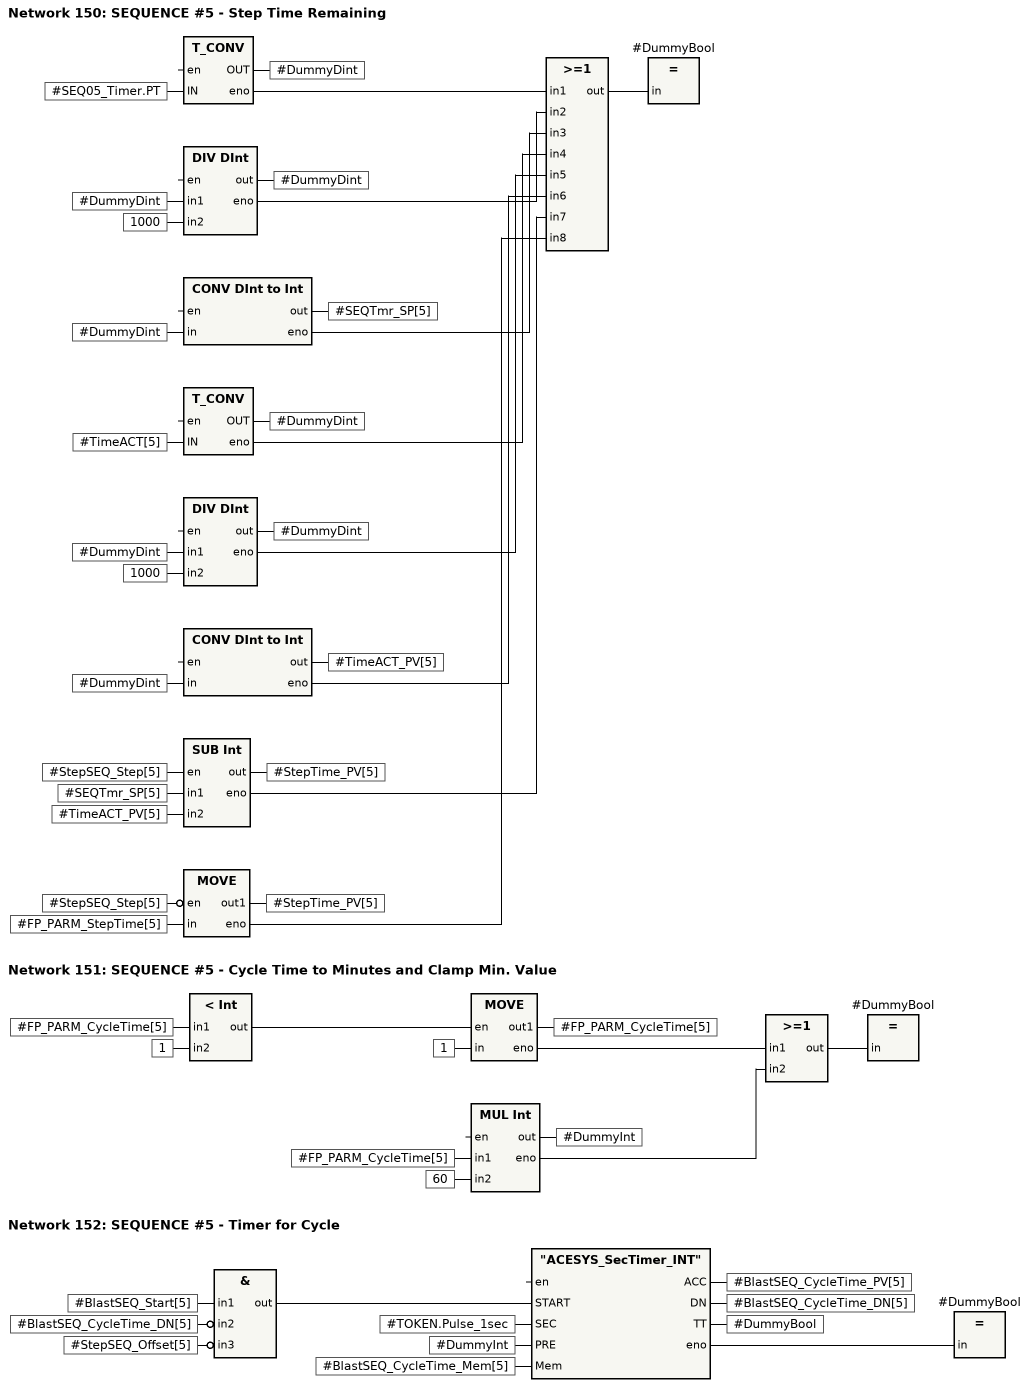
   // ENO of a box is taken as its EN; it also drops when the box reports an error
   #DummyDint := T_CONV(IN := #SEQ05_Timer.PT);
   #DummyDint := #DummyDint / 1000;
   #SEQTmr_SP[5] := DINT_TO_INT(#DummyDint);
   #DummyDint := T_CONV(IN := #TimeACT[5]);
   #DummyDint := #DummyDint / 1000;
   #TimeACT_PV[5] := DINT_TO_INT(#DummyDint);
   IF #StepSEQ_Step[5] THEN #StepTime_PV[5] := #SEQTmr_SP[5] - #TimeACT_PV[5]; END_IF;
   IF NOT #StepSEQ_Step[5] THEN #StepTime_PV[5] := #FP_PARM_StepTime[5]; END_IF;
   #DummyBool := TRUE OR TRUE OR TRUE OR TRUE OR TRUE OR TRUE OR #StepSEQ_Step[5] OR NOT #StepSEQ_Step[5];
END_REGION

REGION Network 151: SEQUENCE #5 - Cycle Time to Minutes and Clamp Min. Value
   // ENO of a box is taken as its EN; it also drops when the box reports an error
   #_w1 := #FP_PARM_CycleTime[5] < 1;
   IF #_w1 THEN #FP_PARM_CycleTime[5] := 1; END_IF;
   #DummyInt := #FP_PARM_CycleTime[5] * 60;
   #DummyBool := #_w1 OR TRUE;
END_REGION

REGION Network 152: SEQUENCE #5 - Timer for Cycle
   "ACESYS_SecTimer_INT"(START := #BlastSEQ_Start[5] AND NOT #BlastSEQ_CycleTime_DN[5] AND NOT #StepSEQ_Offset[5],
                         SEC := #TOKEN.Pulse_1sec,
                         PRE := #DummyInt,
                         Mem := #BlastSEQ_CycleTime_Mem[5],
                         ACC => #BlastSEQ_CycleTime_PV[5],
                         DN => #BlastSEQ_CycleTime_DN[5],
                         TT => #DummyBool,
                         ENO => #_w1);
   #DummyBool := #_w1;
END_REGION

REGION Network 153: SEQUENCE #6 - Enable and Start
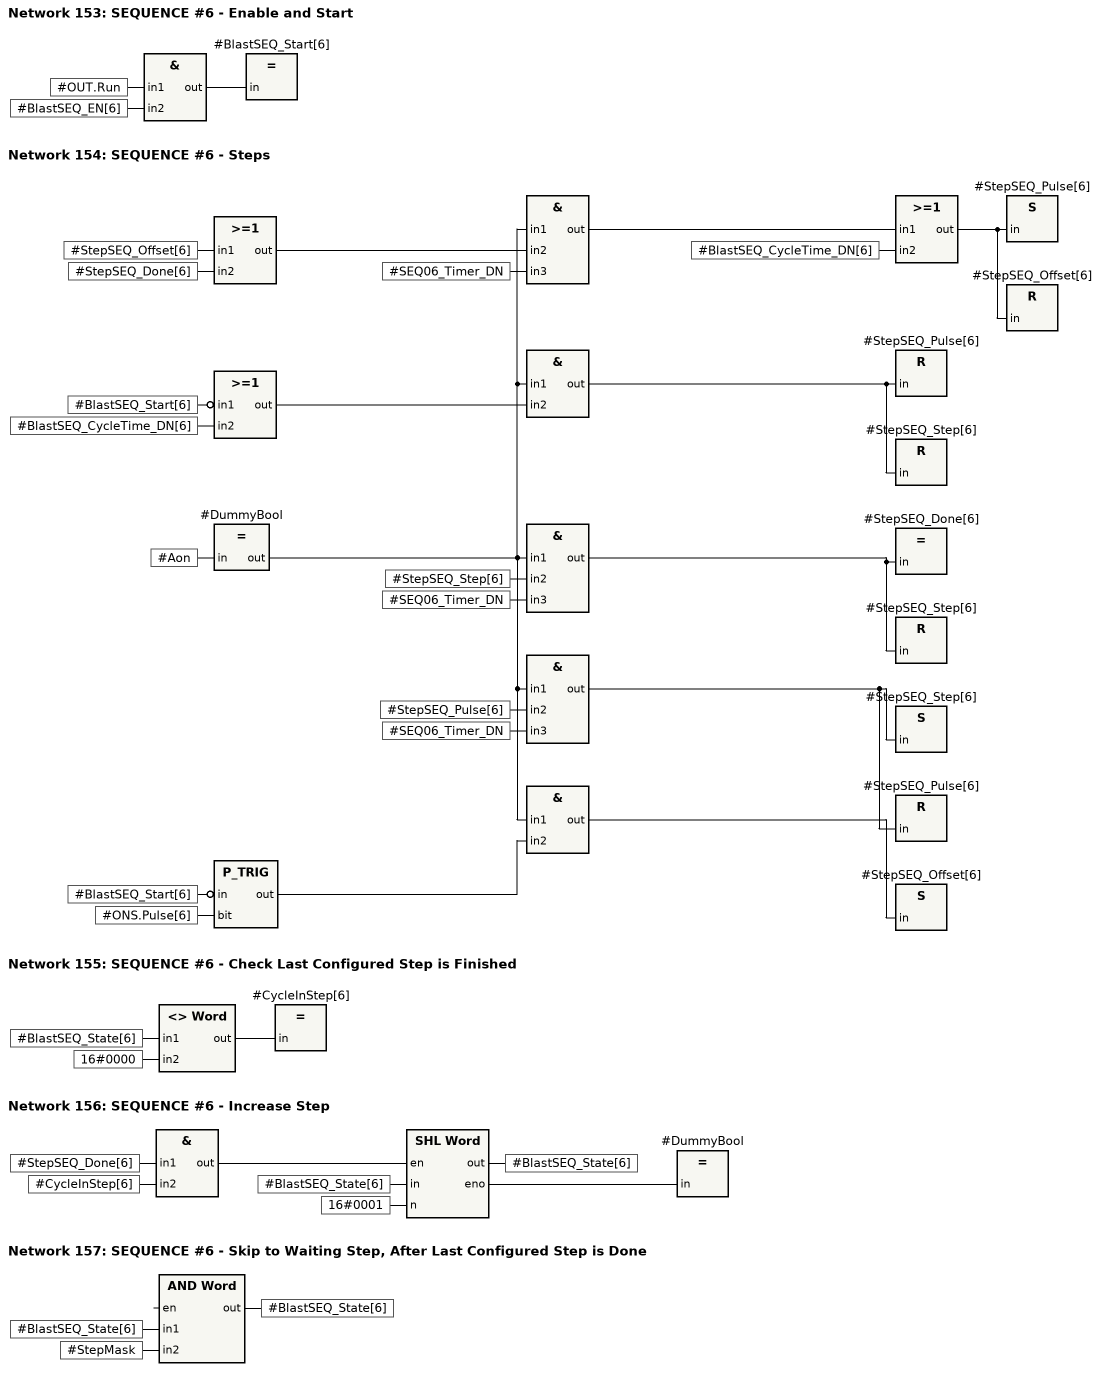
   #BlastSEQ_Start[6] := #OUT.Run AND #BlastSEQ_EN[6];
END_REGION

REGION Network 154: SEQUENCE #6 - Steps
   // Build 002 - 25.Apr.2020 (MIA-US): Replace timer's Q output with tag
   // 
   // ***
   // SEQUENCE 06 LOGIC
   // ***
   // 
   // ***Blaster Sequence***
   // 16#0001 = BQ01
   // 16#0002 = BQ02
   //   -||-
   // 16#4000 = BQ15
   // 16#8000 = BQ16
   // 16#0000 = Cycle Time
   // 
   // ***Step Sequence***
   // - Offset Time
   // - Pulse Time
   // - Step Time
   // - Step Completed
   #DummyBool := #Aon;
   IF #Aon AND (NOT #BlastSEQ_Start[6] OR #BlastSEQ_CycleTime_DN[6]) THEN
       #StepSEQ_Pulse[6] := FALSE;
       #StepSEQ_Step[6] := FALSE;
   END_IF;
   #StepSEQ_Done[6] := #Aon AND #StepSEQ_Step[6] AND #SEQ06_Timer_DN;
   IF #Aon AND #StepSEQ_Step[6] AND #SEQ06_Timer_DN THEN #StepSEQ_Step[6] := FALSE; END_IF;
   IF #Aon AND #StepSEQ_Pulse[6] AND #SEQ06_Timer_DN THEN
       #StepSEQ_Step[6] := TRUE;
       #StepSEQ_Pulse[6] := FALSE;
   END_IF;
   IF (#Aon AND (#StepSEQ_Offset[6] OR #StepSEQ_Done[6]) AND #SEQ06_Timer_DN) OR #BlastSEQ_CycleTime_DN[6] THEN
       #StepSEQ_Pulse[6] := TRUE;
       #StepSEQ_Offset[6] := FALSE;
   END_IF;
   #_w1 := NOT #BlastSEQ_Start[6] AND NOT #ONS.Pulse[6];   // rising edge
   #ONS.Pulse[6] := NOT #BlastSEQ_Start[6];
   IF #Aon AND #_w1 THEN #StepSEQ_Offset[6] := TRUE; END_IF;
END_REGION

REGION Network 155: SEQUENCE #6 - Check Last Configured Step is Finished
   // 16#0000 is the waiting state
   #CycleInStep[6] := #BlastSEQ_State[6] <> 16#0000;
END_REGION

REGION Network 156: SEQUENCE #6 - Increase Step
   // Set next step by shifting one bit to the left in the sequence status
   // ENO of a box is taken as its EN; it also drops when the box reports an error
   #_w1 := #StepSEQ_Done[6] AND #CycleInStep[6];
   IF #_w1 THEN #BlastSEQ_State[6] := SHL(IN := #BlastSEQ_State[6], N := 16#0001); END_IF;
   #DummyBool := #_w1;
END_REGION

REGION Network 157: SEQUENCE #6 - Skip to Waiting Step, After Last Configured Step is Done
   // Sequence Status will become 16#0000 once the shifting bit moves into the unconfigured steps (0 in Step Mask)
   #BlastSEQ_State[6] := #BlastSEQ_State[6] AND #StepMask;
END_REGION

REGION Network 158: SEQUENCE #6 - Offset Step
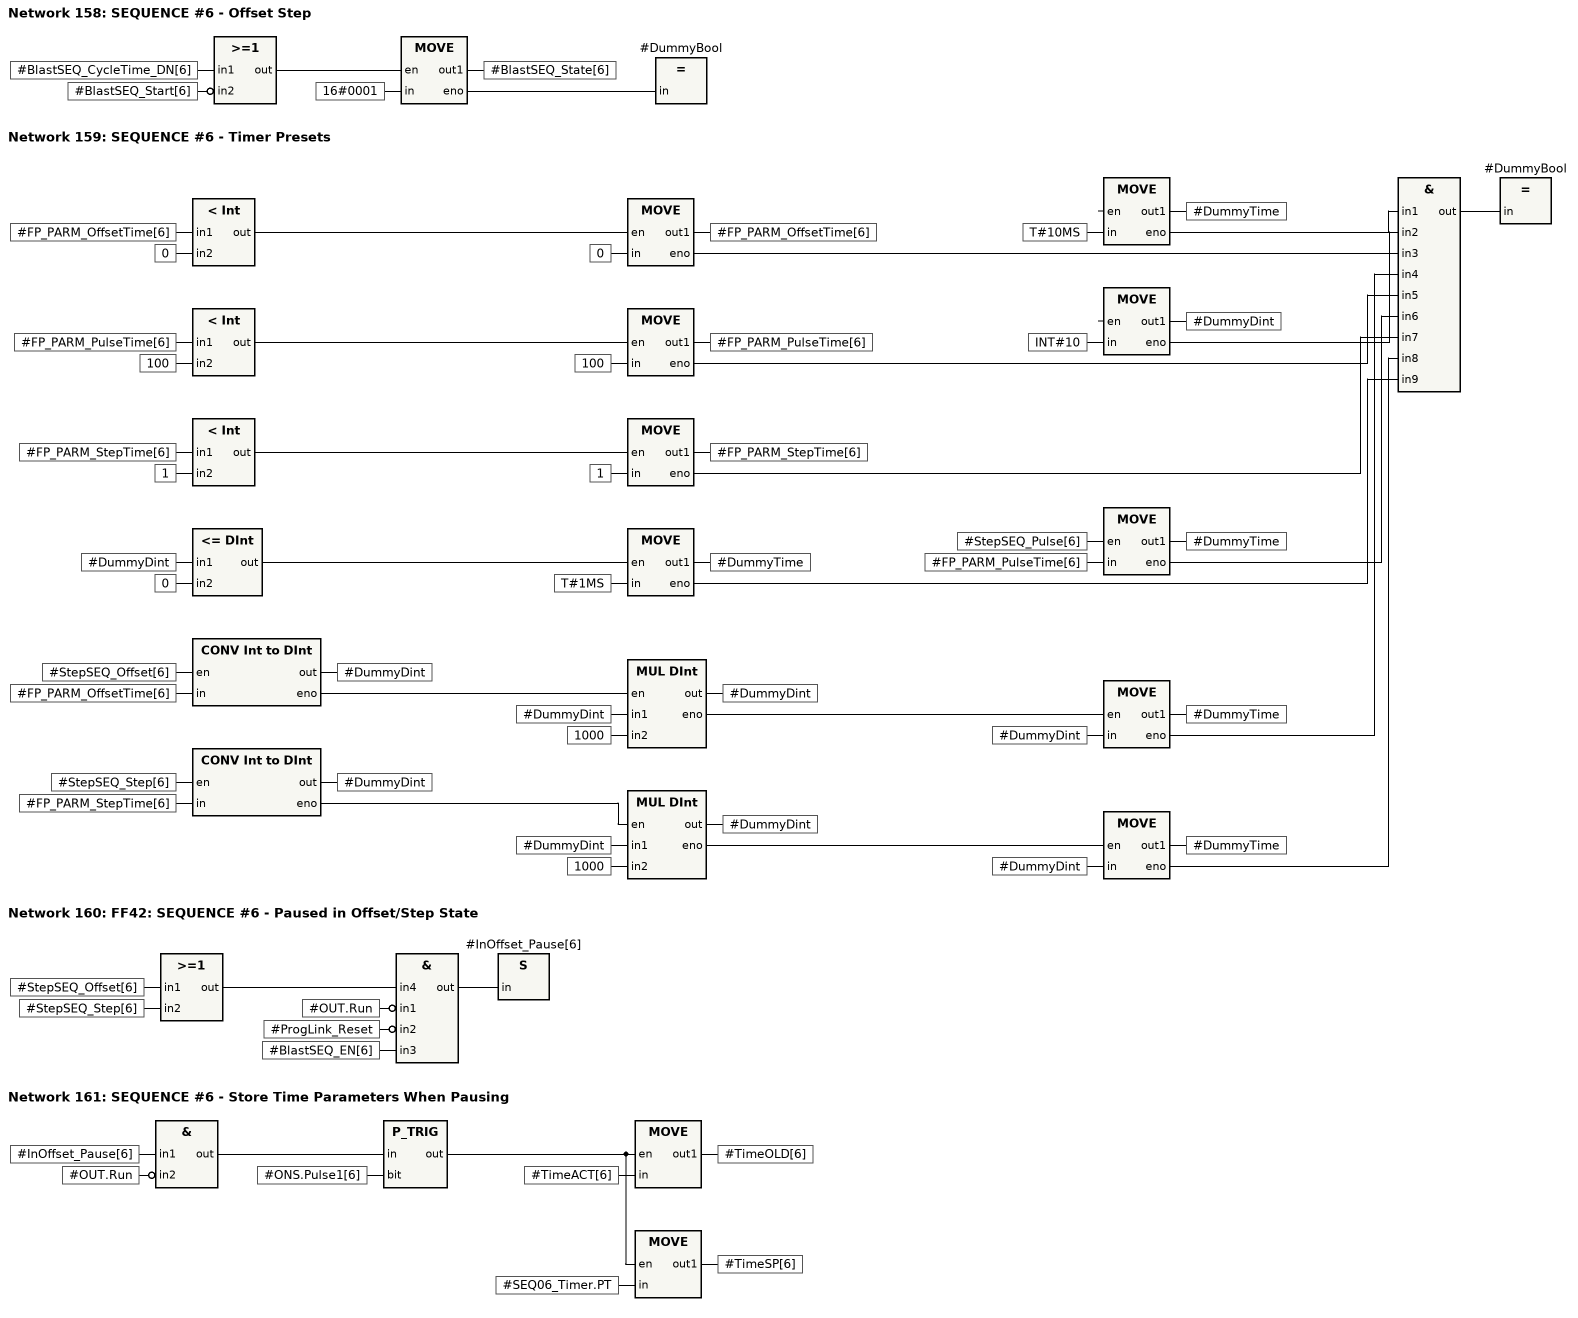
   // ENO of a box is taken as its EN; it also drops when the box reports an error
   #_w1 := #BlastSEQ_CycleTime_DN[6] OR NOT #BlastSEQ_Start[6];
   IF #_w1 THEN #BlastSEQ_State[6] := 16#0001; END_IF;
   #DummyBool := #_w1;
END_REGION

REGION Network 159: SEQUENCE #6 - Timer Presets
   // *Convert Offset Time to minutes and clamp minimum value
   // 
   // *Convert Pulse Time to ms and clamp minimum value
   // 
   // *Convert Step Time to seconds and clamp minimum value
   // ENO of a box is taken as its EN; it also drops when the box reports an error
   #DummyTime := T#10MS;
   #DummyDint := INT#10;
   #_w1 := #FP_PARM_OffsetTime[6] < 0;
   IF #_w1 THEN #FP_PARM_OffsetTime[6] := 0; END_IF;
   IF #StepSEQ_Offset[6] THEN
       #DummyDint := INT_TO_DINT(#FP_PARM_OffsetTime[6]);
       #DummyDint := #DummyDint * 1000;
       #DummyTime := #DummyDint;
   END_IF;
   #_w2 := #FP_PARM_PulseTime[6] < 100;
   IF #_w2 THEN #FP_PARM_PulseTime[6] := 100; END_IF;
   IF #StepSEQ_Pulse[6] THEN #DummyTime := #FP_PARM_PulseTime[6]; END_IF;
   #_w3 := #FP_PARM_StepTime[6] < 1;
   IF #_w3 THEN #FP_PARM_StepTime[6] := 1; END_IF;
   IF #StepSEQ_Step[6] THEN
       #DummyDint := INT_TO_DINT(#FP_PARM_StepTime[6]);
       #DummyDint := #DummyDint * 1000;
       #DummyTime := #DummyDint;
   END_IF;
   #_w4 := #DummyDint <= 0;
   IF #_w4 THEN #DummyTime := T#1MS; END_IF;
   #DummyBool := #_w1 AND #StepSEQ_Offset[6] AND #_w2 AND #StepSEQ_Pulse[6] AND #_w3 AND #StepSEQ_Step[6] AND #_w4;
END_REGION

REGION Network 160: FF42: SEQUENCE #6 - Paused in Offset/Step State
   FF42:
   IF (#StepSEQ_Offset[6] OR #StepSEQ_Step[6]) AND NOT #OUT.Run AND NOT #ProgLink_Reset AND #BlastSEQ_EN[6] THEN
       #InOffset_Pause[6] := TRUE;
   END_IF;
END_REGION

REGION Network 161: SEQUENCE #6 - Store Time Parameters When Pausing
   #_w1 := #InOffset_Pause[6] AND NOT #OUT.Run;
   #_w2 := #_w1 AND NOT #ONS.Pulse1[6];   // rising edge
   #ONS.Pulse1[6] := #_w1;
   IF #_w2 THEN
       #TimeOLD[6] := #TimeACT[6];
       #TimeSP[6] := #SEQ06_Timer.PT;
   END_IF;
END_REGION

REGION Network 162: SEQUENCE #6 - Calculate Time Remaining When Pausing
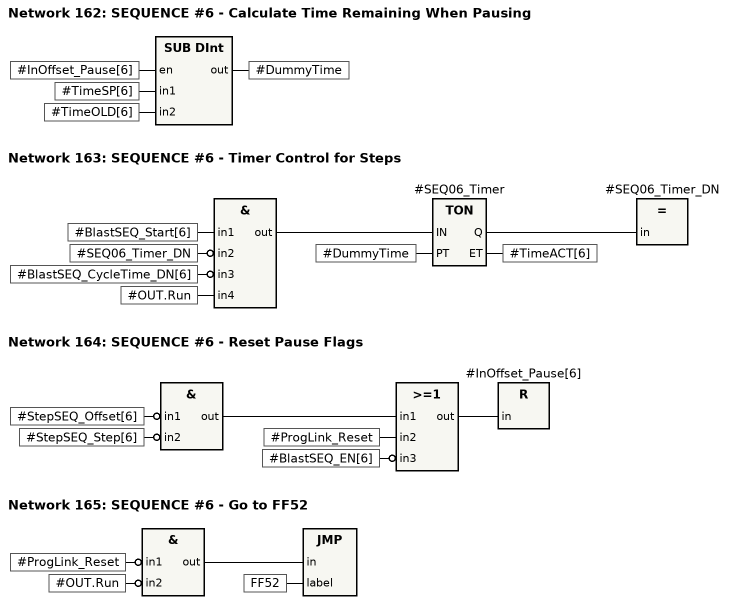
   IF #InOffset_Pause[6] THEN #DummyTime := #TimeSP[6] - #TimeOLD[6]; END_IF;
END_REGION

REGION Network 163: SEQUENCE #6 - Timer Control for Steps
   // Build 002 - 25.Apr.2020 (MIA-US): Added tag to timer's Q output.
   // -Offset time
   // -Pulse time
   // -Step time
   #SEQ06_Timer(IN := #BlastSEQ_Start[6] AND NOT #SEQ06_Timer_DN AND NOT #BlastSEQ_CycleTime_DN[6] AND #OUT.Run,   // TON
                PT := #DummyTime,
                ET => #TimeACT[6]);
   #SEQ06_Timer_DN := #SEQ06_Timer.Q;
END_REGION

REGION Network 164: SEQUENCE #6 - Reset Pause Flags
   IF (NOT #StepSEQ_Offset[6] AND NOT #StepSEQ_Step[6]) OR #ProgLink_Reset OR NOT #BlastSEQ_EN[6] THEN
       #InOffset_Pause[6] := FALSE;
   END_IF;
END_REGION

REGION Network 165: SEQUENCE #6 - Go to FF52
   IF NOT #ProgLink_Reset AND NOT #OUT.Run THEN GOTO FF52; END_IF;
END_REGION

REGION Network 166: SEQUENCE #6 - Step Time Remaining
   // Display countdown in seconds for active step
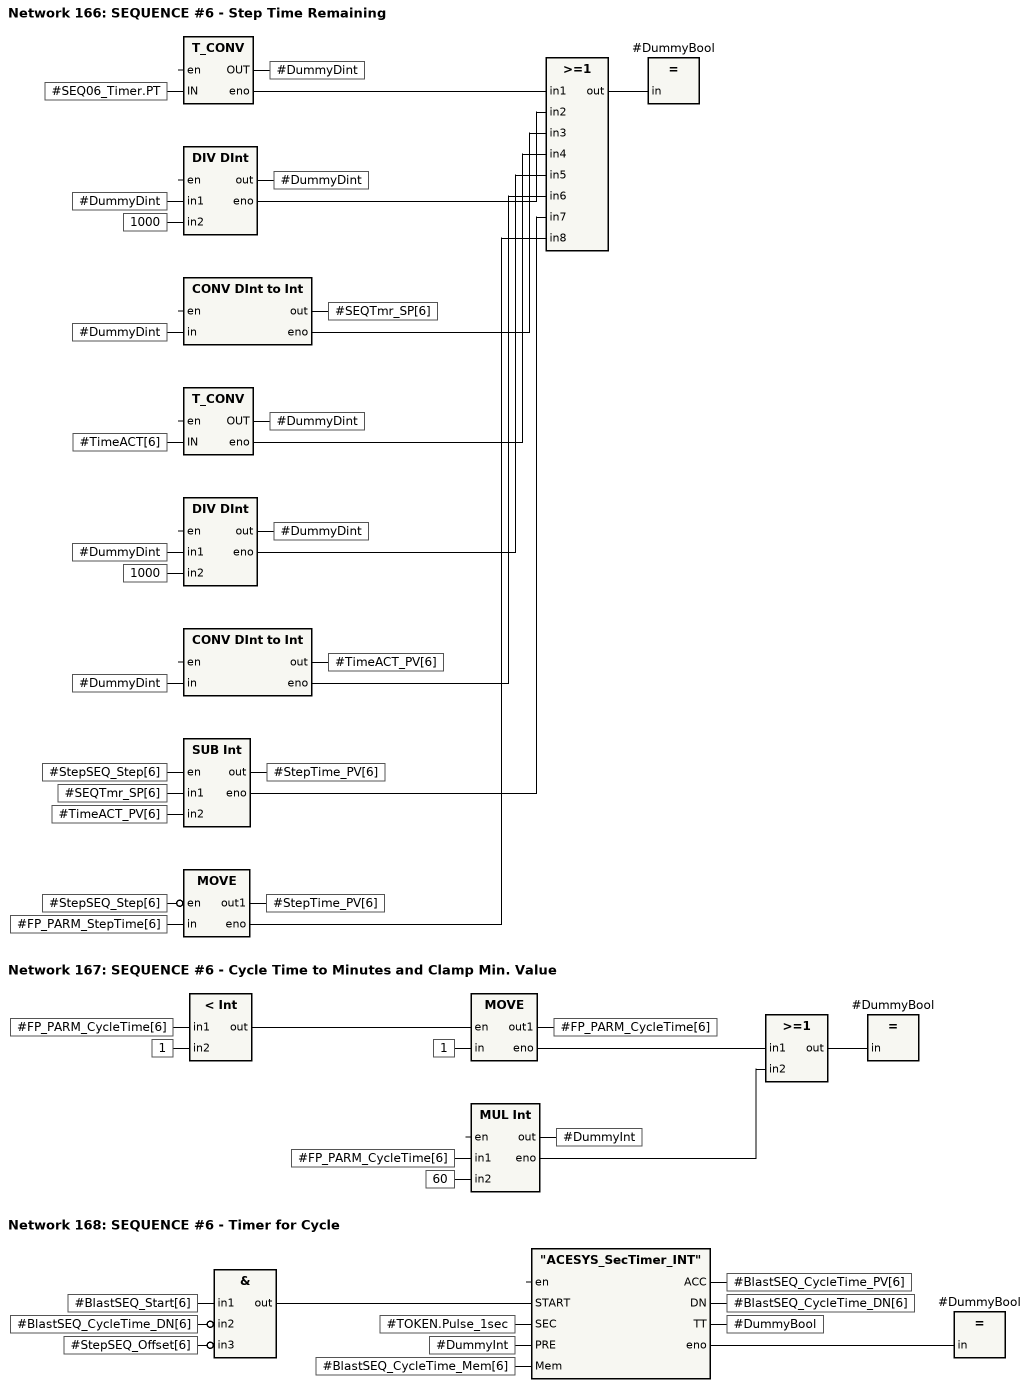
   // ENO of a box is taken as its EN; it also drops when the box reports an error
   #DummyDint := T_CONV(IN := #SEQ06_Timer.PT);
   #DummyDint := #DummyDint / 1000;
   #SEQTmr_SP[6] := DINT_TO_INT(#DummyDint);
   #DummyDint := T_CONV(IN := #TimeACT[6]);
   #DummyDint := #DummyDint / 1000;
   #TimeACT_PV[6] := DINT_TO_INT(#DummyDint);
   IF #StepSEQ_Step[6] THEN #StepTime_PV[6] := #SEQTmr_SP[6] - #TimeACT_PV[6]; END_IF;
   IF NOT #StepSEQ_Step[6] THEN #StepTime_PV[6] := #FP_PARM_StepTime[6]; END_IF;
   #DummyBool := TRUE OR TRUE OR TRUE OR TRUE OR TRUE OR TRUE OR #StepSEQ_Step[6] OR NOT #StepSEQ_Step[6];
END_REGION

REGION Network 167: SEQUENCE #6 - Cycle Time to Minutes and Clamp Min. Value
   // ENO of a box is taken as its EN; it also drops when the box reports an error
   #_w1 := #FP_PARM_CycleTime[6] < 1;
   IF #_w1 THEN #FP_PARM_CycleTime[6] := 1; END_IF;
   #DummyInt := #FP_PARM_CycleTime[6] * 60;
   #DummyBool := #_w1 OR TRUE;
END_REGION

REGION Network 168: SEQUENCE #6 - Timer for Cycle
   "ACESYS_SecTimer_INT"(START := #BlastSEQ_Start[6] AND NOT #BlastSEQ_CycleTime_DN[6] AND NOT #StepSEQ_Offset[6],
                         SEC := #TOKEN.Pulse_1sec,
                         PRE := #DummyInt,
                         Mem := #BlastSEQ_CycleTime_Mem[6],
                         ACC => #BlastSEQ_CycleTime_PV[6],
                         DN => #BlastSEQ_CycleTime_DN[6],
                         TT => #DummyBool,
                         ENO => #_w1);
   #DummyBool := #_w1;
END_REGION

REGION Network 169: FF52: Initialize ChangeConfig Loop
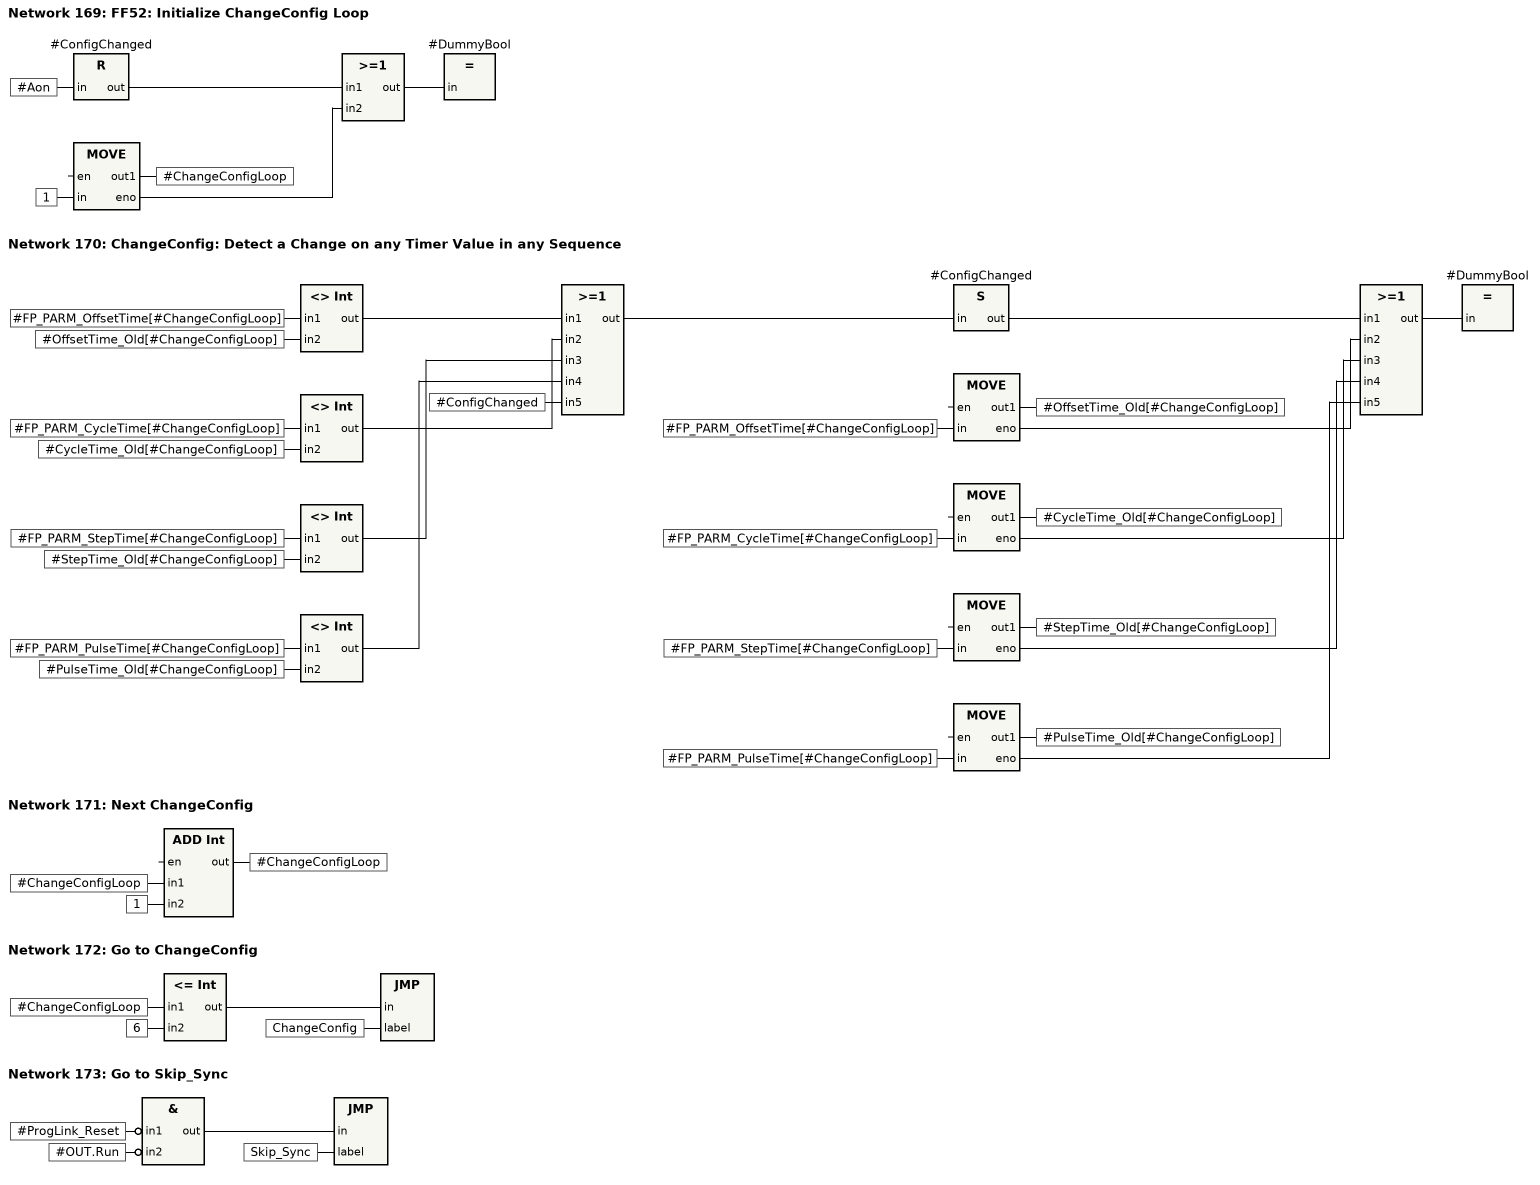
   FF52:
   IF #Aon THEN #ConfigChanged := FALSE; END_IF;
   #ChangeConfigLoop := 1;
   #DummyBool := #Aon OR TRUE;
END_REGION

REGION Network 170: ChangeConfig: Detect a Change on any Timer Value in any Sequence
   ChangeConfig:
   #_w1 := (#FP_PARM_OffsetTime[#ChangeConfigLoop] <> #OffsetTime_Old[#ChangeConfigLoop]) OR (#FP_PARM_CycleTime[#ChangeConfigLoop] <> #CycleTime_Old[#ChangeConfigLoop]) OR (#FP_PARM_StepTime[#ChangeConfigLoop] <> #StepTime_Old[#ChangeConfigLoop]) OR (#FP_PARM_PulseTime[#ChangeConfigLoop] <> #PulseTime_Old[#ChangeConfigLoop]) OR #ConfigChanged;
   IF #_w1 THEN #ConfigChanged := TRUE; END_IF;
   #OffsetTime_Old[#ChangeConfigLoop] := #FP_PARM_OffsetTime[#ChangeConfigLoop];
   #CycleTime_Old[#ChangeConfigLoop] := #FP_PARM_CycleTime[#ChangeConfigLoop];
   #StepTime_Old[#ChangeConfigLoop] := #FP_PARM_StepTime[#ChangeConfigLoop];
   #PulseTime_Old[#ChangeConfigLoop] := #FP_PARM_PulseTime[#ChangeConfigLoop];
   #DummyBool := #_w1 OR TRUE OR TRUE OR TRUE OR TRUE;
END_REGION

REGION Network 171: Next ChangeConfig
   #ChangeConfigLoop := #ChangeConfigLoop + 1;
END_REGION

REGION Network 172: Go to ChangeConfig
   IF #ChangeConfigLoop <= 6 THEN GOTO ChangeConfig; END_IF;
END_REGION

REGION Network 173: Go to Skip_Sync
   IF NOT #ProgLink_Reset AND NOT #OUT.Run THEN GOTO Skip_Sync; END_IF;
END_REGION

REGION Network 174: Sequence Sync Timer Trigger
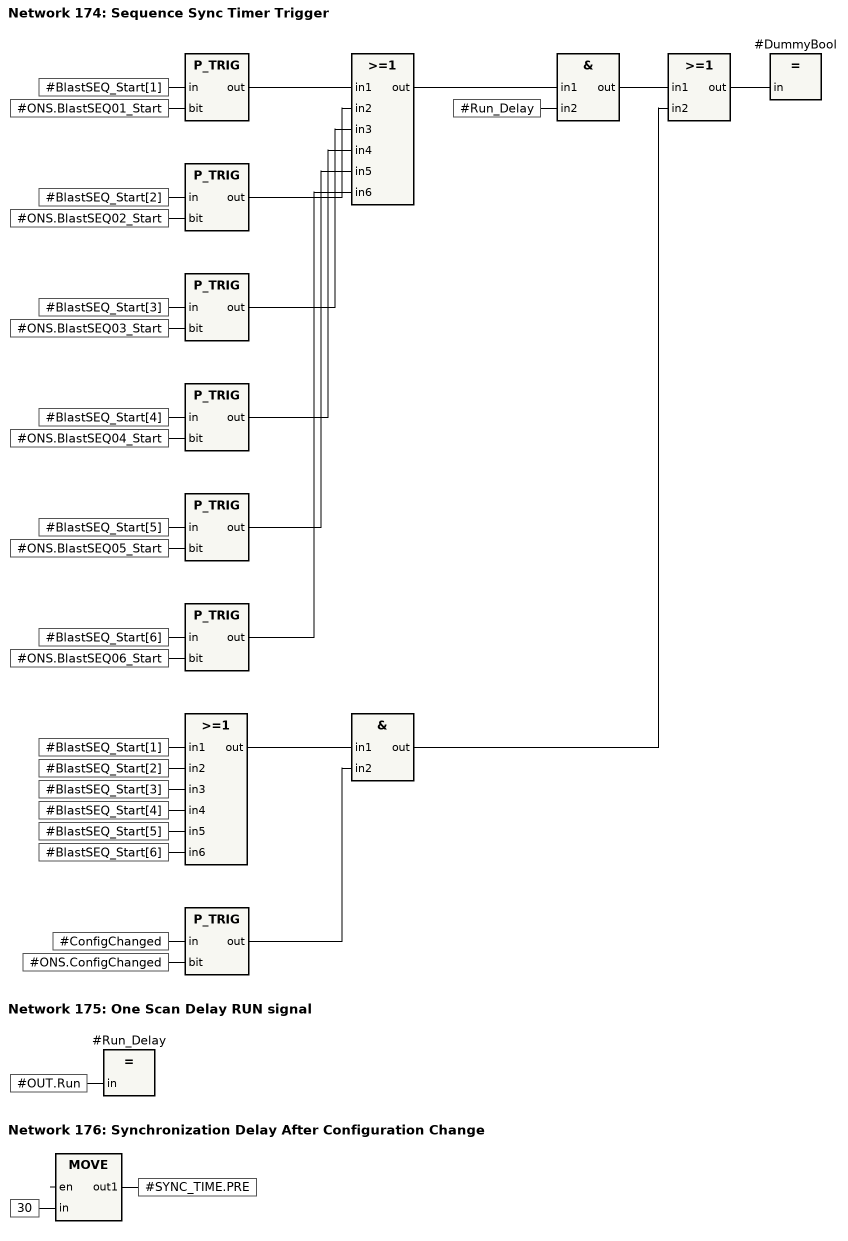
   #_w1 := #BlastSEQ_Start[1] AND NOT #ONS.BlastSEQ01_Start;   // rising edge
   #ONS.BlastSEQ01_Start := #BlastSEQ_Start[1];
   #_w2 := #BlastSEQ_Start[2] AND NOT #ONS.BlastSEQ02_Start;   // rising edge
   #ONS.BlastSEQ02_Start := #BlastSEQ_Start[2];
   #_w3 := #BlastSEQ_Start[3] AND NOT #ONS.BlastSEQ03_Start;   // rising edge
   #ONS.BlastSEQ03_Start := #BlastSEQ_Start[3];
   #_w4 := #BlastSEQ_Start[4] AND NOT #ONS.BlastSEQ04_Start;   // rising edge
   #ONS.BlastSEQ04_Start := #BlastSEQ_Start[4];
   #_w5 := #BlastSEQ_Start[5] AND NOT #ONS.BlastSEQ05_Start;   // rising edge
   #ONS.BlastSEQ05_Start := #BlastSEQ_Start[5];
   #_w6 := #BlastSEQ_Start[6] AND NOT #ONS.BlastSEQ06_Start;   // rising edge
   #ONS.BlastSEQ06_Start := #BlastSEQ_Start[6];
   #_w7 := #ConfigChanged AND NOT #ONS.ConfigChanged;   // rising edge
   #ONS.ConfigChanged := #ConfigChanged;
   #DummyBool := ((#_w1 OR #_w2 OR #_w3 OR #_w4 OR #_w5 OR #_w6) AND #Run_Delay) OR ((#BlastSEQ_Start[1] OR #BlastSEQ_Start[2] OR #BlastSEQ_Start[3] OR #BlastSEQ_Start[4] OR #BlastSEQ_Start[5] OR #BlastSEQ_Start[6]) AND #_w7);
END_REGION

REGION Network 175: One Scan Delay RUN signal
   #Run_Delay := #OUT.Run;
END_REGION

REGION Network 176: Synchronization Delay After Configuration Change
   // Time After Last Time Change Before Sequences are Re-initialized
   #SYNC_TIME.PRE := 30;
END_REGION

REGION Network 177: Sequence Sync Timer
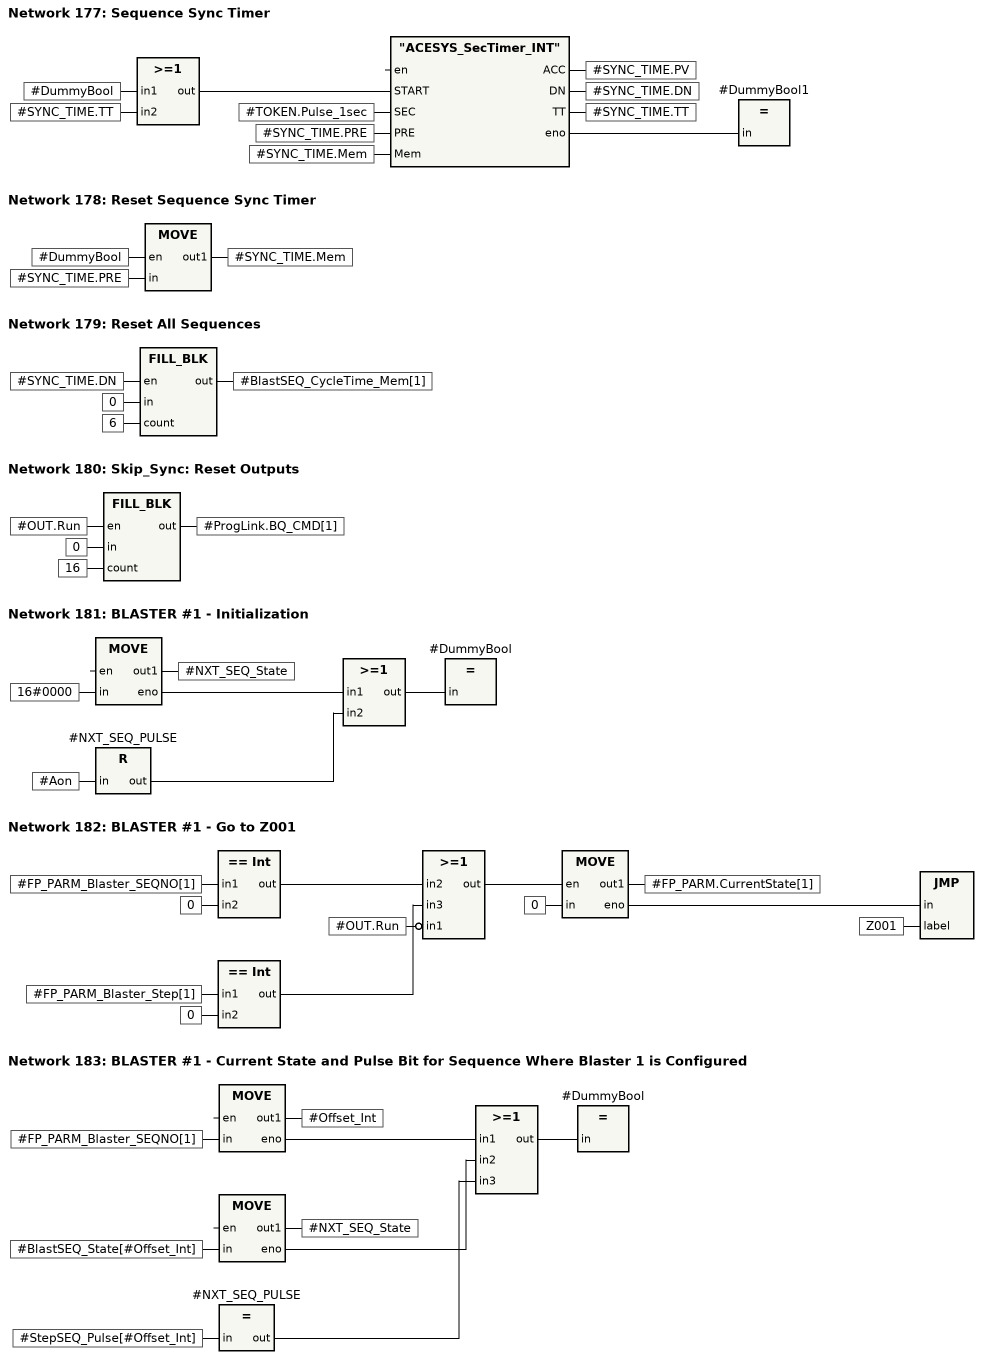
   "ACESYS_SecTimer_INT"(START := #DummyBool OR #SYNC_TIME.TT,
                         SEC := #TOKEN.Pulse_1sec,
                         PRE := #SYNC_TIME.PRE,
                         Mem := #SYNC_TIME.Mem,
                         ACC => #SYNC_TIME.PV,
                         DN => #SYNC_TIME.DN,
                         TT => #SYNC_TIME.TT,
                         ENO => #_w1);
   #DummyBool1 := #_w1;
END_REGION

REGION Network 178: Reset Sequence Sync Timer
   // Reset upon a configuration change or a new sequence is started
   IF #DummyBool THEN #SYNC_TIME.Mem := #SYNC_TIME.PRE; END_IF;
END_REGION

REGION Network 179: Reset All Sequences
   IF #SYNC_TIME.DN THEN FILL_BLK(IN := 0, COUNT := 6, OUT => #BlastSEQ_CycleTime_Mem[1]); END_IF;
END_REGION

REGION Network 180: Skip_Sync: Reset Outputs
   // Build 002 - 25.Apr.2020 (MIA-US): Added enable to prevent clearing blasters command data from other programs when not running
   Skip_Sync:
   IF #OUT.Run THEN FILL_BLK(IN := 0, COUNT := 16, OUT => #ProgLink.BQ_CMD[1]); END_IF;
END_REGION

REGION Network 181: BLASTER #1 - Initialization
   #NXT_SEQ_State := 16#0000;
   IF #Aon THEN #NXT_SEQ_PULSE := FALSE; END_IF;
   #DummyBool := TRUE OR #Aon;
END_REGION

REGION Network 182: BLASTER #1 - Go to Z001
   // If Blaster #1 is not configured in any sequence/step then clear state and go to next blaster
   #_w1 := (#FP_PARM_Blaster_SEQNO[1] = 0) OR (#FP_PARM_Blaster_Step[1] = 0) OR NOT #OUT.Run;
   IF #_w1 THEN
       #FP_PARM.CurrentState[1] := 0;
       GOTO Z001;
   END_IF;
END_REGION

REGION Network 183: BLASTER #1 - Current State and Pulse Bit for Sequence Where Blaster 1 is Configured
   #Offset_Int := #FP_PARM_Blaster_SEQNO[1];
   #NXT_SEQ_State := #BlastSEQ_State[#Offset_Int];
   #NXT_SEQ_PULSE := #StepSEQ_Pulse[#Offset_Int];
   #DummyBool := TRUE OR TRUE OR #StepSEQ_Pulse[#Offset_Int];
END_REGION

REGION Network 184: BLASTER #1 - Go to Skip_Exp1
   // Exceptions: 
   // 16#0000: Log(0) is not possible
   // 16#8000: Bit 15 is INT bit sign
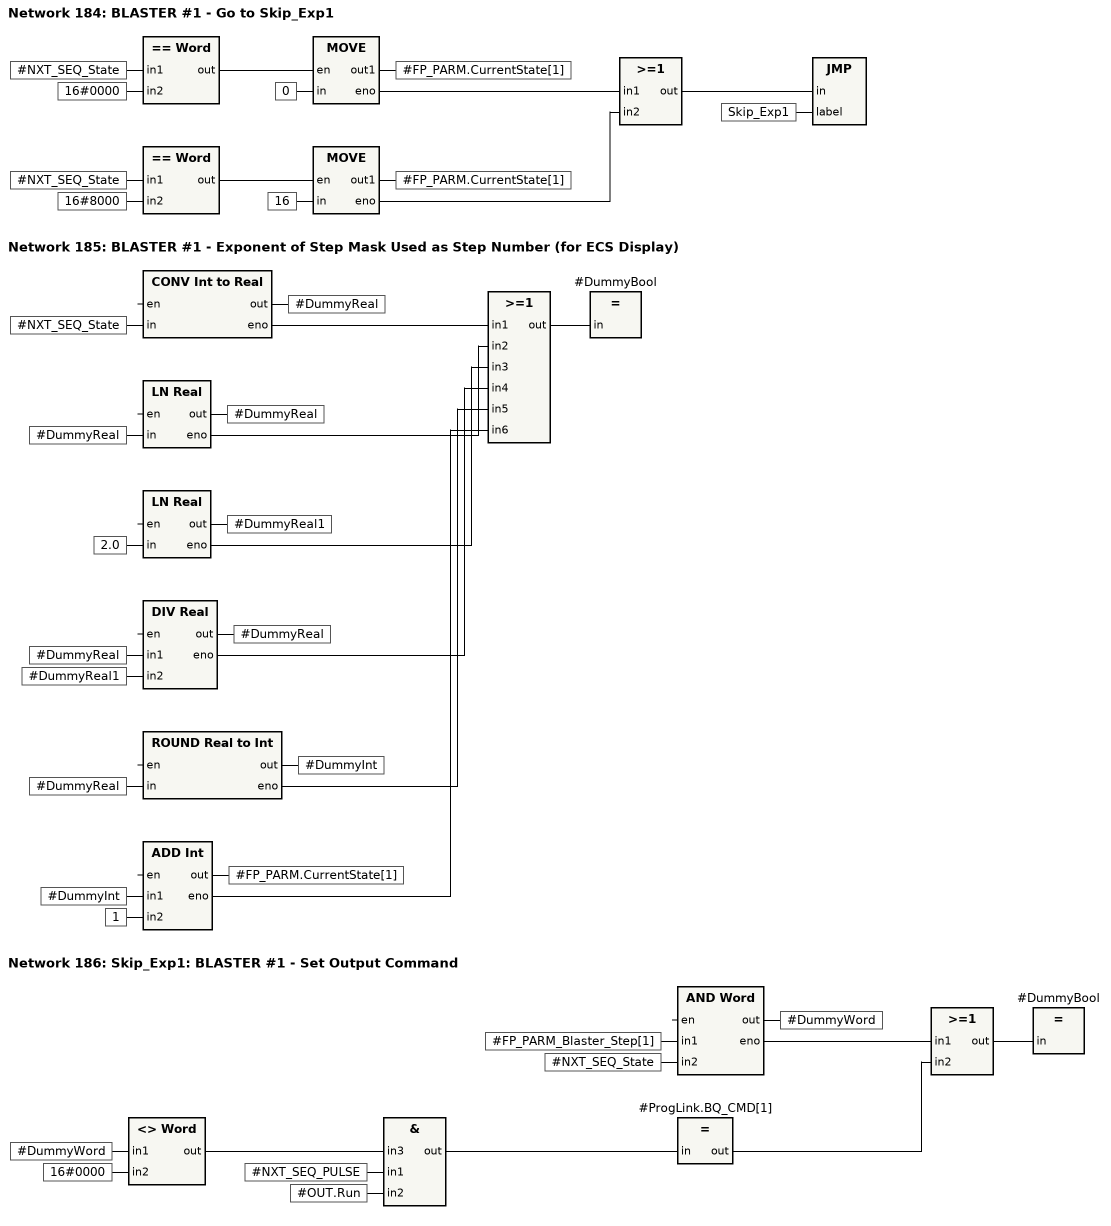
   #_w1 := #NXT_SEQ_State = 16#0000;
   IF #_w1 THEN #FP_PARM.CurrentState[1] := 0; END_IF;
   #_w2 := #NXT_SEQ_State = 16#8000;
   IF #_w2 THEN #FP_PARM.CurrentState[1] := 16; END_IF;
   IF #_w1 OR #_w2 THEN GOTO Skip_Exp1; END_IF;
END_REGION

REGION Network 185: BLASTER #1 - Exponent of Step Mask Used as Step Number (for ECS Display)
   // Step Number = [ln(NXT_SEQ_State)/ln(2)]+1
   #DummyReal := INT_TO_REAL(#NXT_SEQ_State);
   #DummyReal := LN(#DummyReal);
   #DummyReal1 := LN(2.0);
   #DummyReal := #DummyReal / #DummyReal1;
   #DummyInt := ROUND(#DummyReal);
   #FP_PARM.CurrentState[1] := #DummyInt + 1;
   #DummyBool := TRUE OR TRUE OR TRUE OR TRUE OR TRUE OR TRUE;
END_REGION

REGION Network 186: Skip_Exp1: BLASTER #1 - Set Output Command
   Skip_Exp1:
   #DummyWord := #FP_PARM_Blaster_Step[1] AND #NXT_SEQ_State;
   #ProgLink.BQ_CMD[1] := (#DummyWord <> 16#0000) AND #NXT_SEQ_PULSE AND #OUT.Run;
   #DummyBool := TRUE OR ((#DummyWord <> 16#0000) AND #NXT_SEQ_PULSE AND #OUT.Run);
END_REGION

REGION Network 187: Z001: BLASTER #2 - Initialization
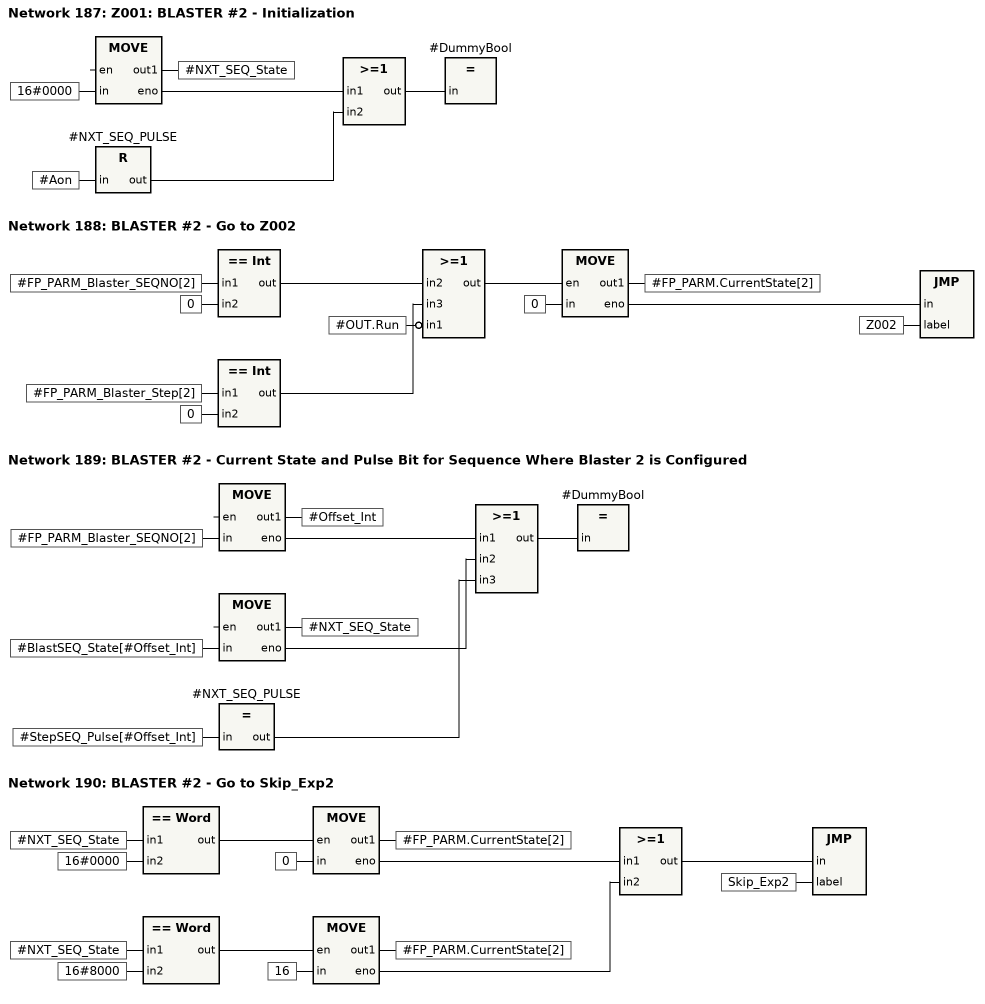
   Z001:
   #NXT_SEQ_State := 16#0000;
   IF #Aon THEN #NXT_SEQ_PULSE := FALSE; END_IF;
   #DummyBool := TRUE OR #Aon;
END_REGION

REGION Network 188: BLASTER #2 - Go to Z002
   // If Blaster #2 is not configured in any sequence/step then clear state and go to next blaster
   #_w1 := (#FP_PARM_Blaster_SEQNO[2] = 0) OR (#FP_PARM_Blaster_Step[2] = 0) OR NOT #OUT.Run;
   IF #_w1 THEN
       #FP_PARM.CurrentState[2] := 0;
       GOTO Z002;
   END_IF;
END_REGION

REGION Network 189: BLASTER #2 - Current State and Pulse Bit for Sequence Where Blaster 2 is Configured
   #Offset_Int := #FP_PARM_Blaster_SEQNO[2];
   #NXT_SEQ_State := #BlastSEQ_State[#Offset_Int];
   #NXT_SEQ_PULSE := #StepSEQ_Pulse[#Offset_Int];
   #DummyBool := TRUE OR TRUE OR #StepSEQ_Pulse[#Offset_Int];
END_REGION

REGION Network 190: BLASTER #2 - Go to Skip_Exp2
   // Exceptions: 
   // 16#0000: Log(0) is not possible
   // 16#8000: Bit 15 is INT bit sign
   #_w1 := #NXT_SEQ_State = 16#0000;
   IF #_w1 THEN #FP_PARM.CurrentState[2] := 0; END_IF;
   #_w2 := #NXT_SEQ_State = 16#8000;
   IF #_w2 THEN #FP_PARM.CurrentState[2] := 16; END_IF;
   IF #_w1 OR #_w2 THEN GOTO Skip_Exp2; END_IF;
END_REGION

REGION Network 191: BLASTER #2 - Exponent of Step Mask Used as Step Number (for ECS Display)
   // Step Number = [ln(NXT_SEQ_State)/ln(2)]+1
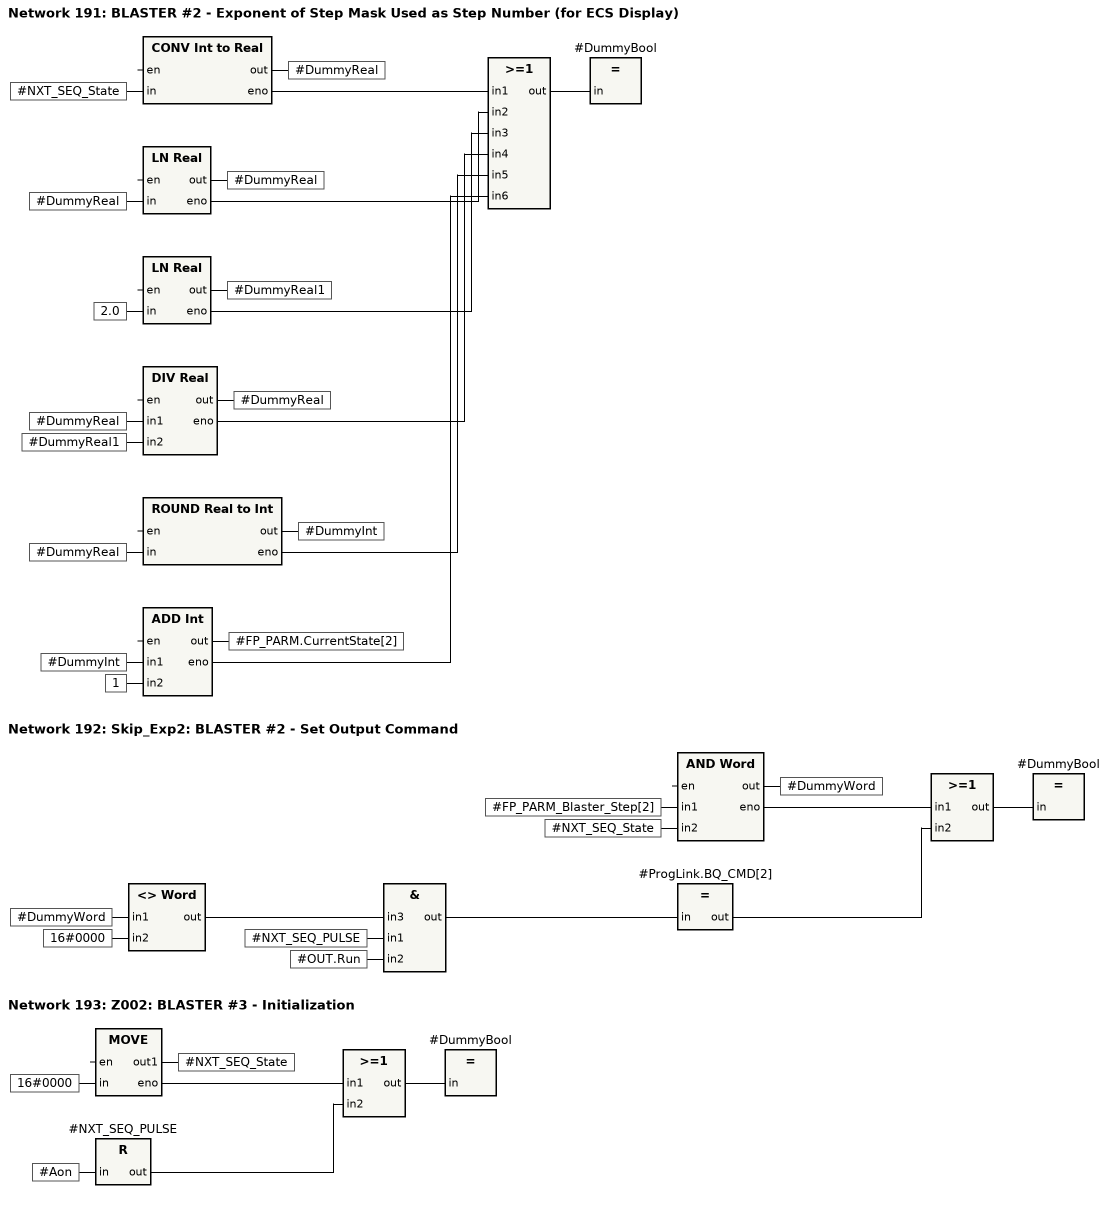
   #DummyReal := INT_TO_REAL(#NXT_SEQ_State);
   #DummyReal := LN(#DummyReal);
   #DummyReal1 := LN(2.0);
   #DummyReal := #DummyReal / #DummyReal1;
   #DummyInt := ROUND(#DummyReal);
   #FP_PARM.CurrentState[2] := #DummyInt + 1;
   #DummyBool := TRUE OR TRUE OR TRUE OR TRUE OR TRUE OR TRUE;
END_REGION

REGION Network 192: Skip_Exp2: BLASTER #2 - Set Output Command
   Skip_Exp2:
   #DummyWord := #FP_PARM_Blaster_Step[2] AND #NXT_SEQ_State;
   #ProgLink.BQ_CMD[2] := (#DummyWord <> 16#0000) AND #NXT_SEQ_PULSE AND #OUT.Run;
   #DummyBool := TRUE OR ((#DummyWord <> 16#0000) AND #NXT_SEQ_PULSE AND #OUT.Run);
END_REGION

REGION Network 193: Z002: BLASTER #3 - Initialization
   Z002:
   #NXT_SEQ_State := 16#0000;
   IF #Aon THEN #NXT_SEQ_PULSE := FALSE; END_IF;
   #DummyBool := TRUE OR #Aon;
END_REGION

REGION Network 194: BLASTER #3 - Go to Z003
   // If Blaster #3 is not configured in any sequence/step then clear state and go to next blaster
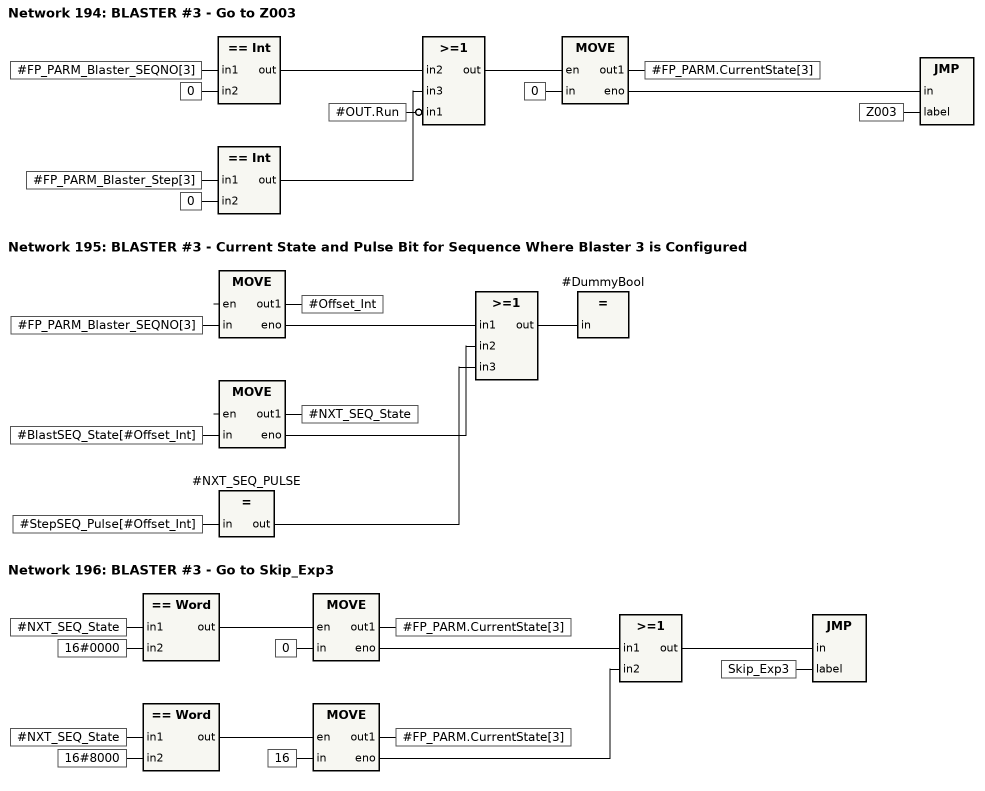
   #_w1 := (#FP_PARM_Blaster_SEQNO[3] = 0) OR (#FP_PARM_Blaster_Step[3] = 0) OR NOT #OUT.Run;
   IF #_w1 THEN
       #FP_PARM.CurrentState[3] := 0;
       GOTO Z003;
   END_IF;
END_REGION

REGION Network 195: BLASTER #3 - Current State and Pulse Bit for Sequence Where Blaster 3 is Configured
   #Offset_Int := #FP_PARM_Blaster_SEQNO[3];
   #NXT_SEQ_State := #BlastSEQ_State[#Offset_Int];
   #NXT_SEQ_PULSE := #StepSEQ_Pulse[#Offset_Int];
   #DummyBool := TRUE OR TRUE OR #StepSEQ_Pulse[#Offset_Int];
END_REGION

REGION Network 196: BLASTER #3 - Go to Skip_Exp3
   // Exceptions: 
   // 16#0000: Log(0) is not possible
   // 16#8000: Bit 15 is INT bit sign
   #_w1 := #NXT_SEQ_State = 16#0000;
   IF #_w1 THEN #FP_PARM.CurrentState[3] := 0; END_IF;
   #_w2 := #NXT_SEQ_State = 16#8000;
   IF #_w2 THEN #FP_PARM.CurrentState[3] := 16; END_IF;
   IF #_w1 OR #_w2 THEN GOTO Skip_Exp3; END_IF;
END_REGION

REGION Network 197: BLASTER #3 - Exponent of Step Mask Used as Step Number (for ECS Display)
   // Step Number = [ln(NXT_SEQ_State)/ln(2)]+1
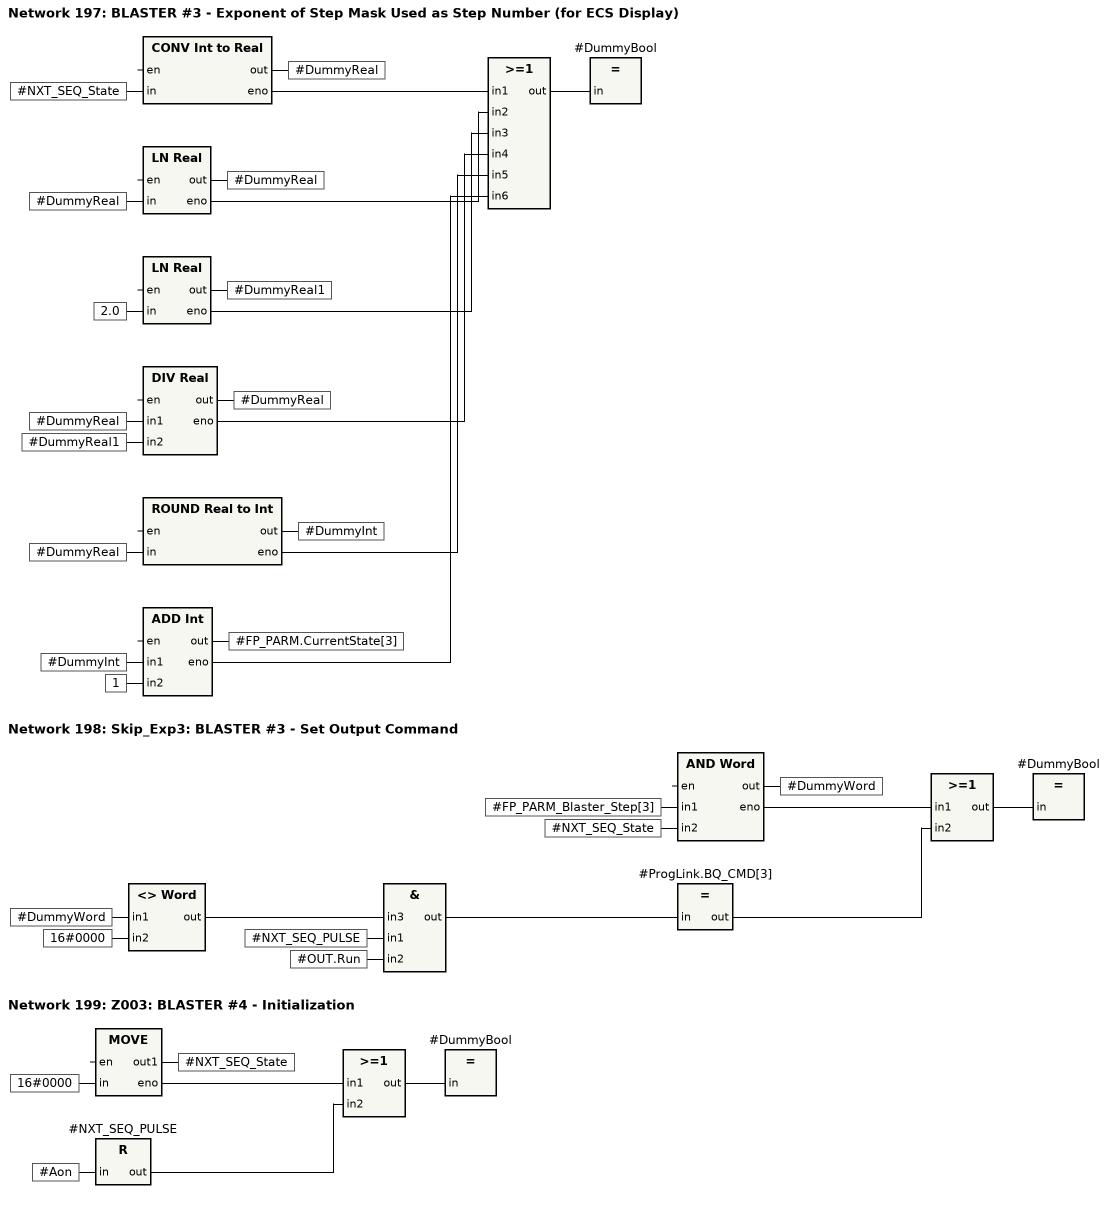
   #DummyReal := INT_TO_REAL(#NXT_SEQ_State);
   #DummyReal := LN(#DummyReal);
   #DummyReal1 := LN(2.0);
   #DummyReal := #DummyReal / #DummyReal1;
   #DummyInt := ROUND(#DummyReal);
   #FP_PARM.CurrentState[3] := #DummyInt + 1;
   #DummyBool := TRUE OR TRUE OR TRUE OR TRUE OR TRUE OR TRUE;
END_REGION

REGION Network 198: Skip_Exp3: BLASTER #3 - Set Output Command
   Skip_Exp3:
   #DummyWord := #FP_PARM_Blaster_Step[3] AND #NXT_SEQ_State;
   #ProgLink.BQ_CMD[3] := (#DummyWord <> 16#0000) AND #NXT_SEQ_PULSE AND #OUT.Run;
   #DummyBool := TRUE OR ((#DummyWord <> 16#0000) AND #NXT_SEQ_PULSE AND #OUT.Run);
END_REGION

REGION Network 199: Z003: BLASTER #4 - Initialization
   Z003:
   #NXT_SEQ_State := 16#0000;
   IF #Aon THEN #NXT_SEQ_PULSE := FALSE; END_IF;
   #DummyBool := TRUE OR #Aon;
END_REGION

REGION Network 200: BLASTER #4 - Go to Z004
   // If Blaster #4 is not configured in any sequence/step then clear state and go to next blaster
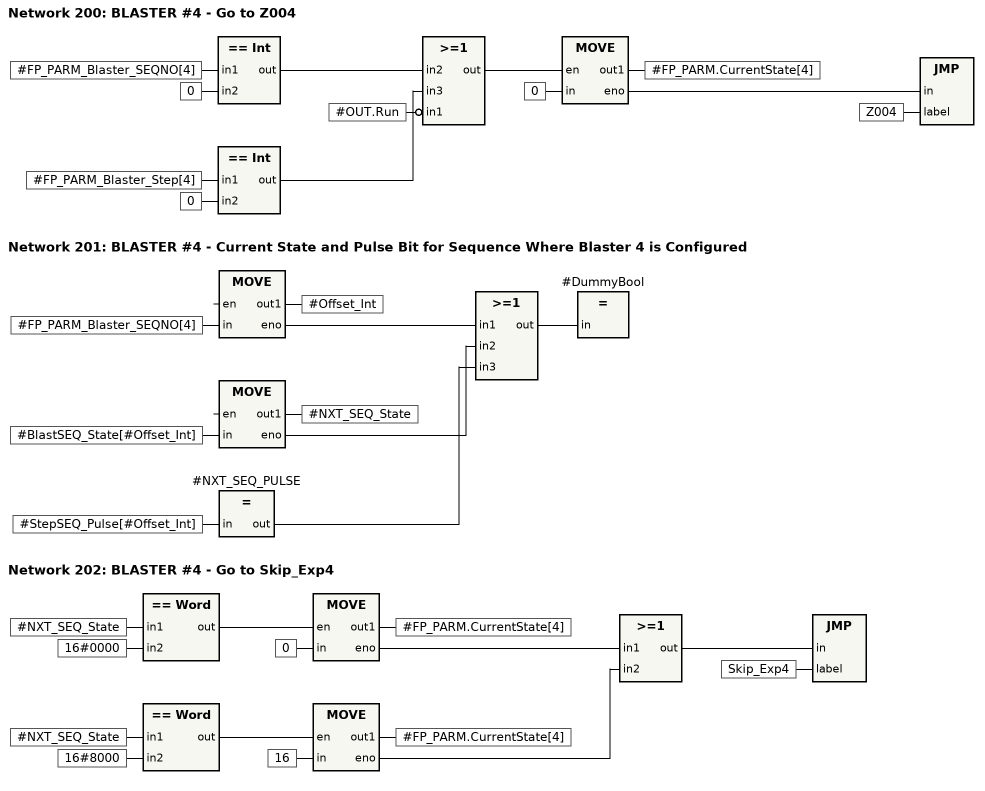
   #_w1 := (#FP_PARM_Blaster_SEQNO[4] = 0) OR (#FP_PARM_Blaster_Step[4] = 0) OR NOT #OUT.Run;
   IF #_w1 THEN
       #FP_PARM.CurrentState[4] := 0;
       GOTO Z004;
   END_IF;
END_REGION

REGION Network 201: BLASTER #4 - Current State and Pulse Bit for Sequence Where Blaster 4 is Configured
   #Offset_Int := #FP_PARM_Blaster_SEQNO[4];
   #NXT_SEQ_State := #BlastSEQ_State[#Offset_Int];
   #NXT_SEQ_PULSE := #StepSEQ_Pulse[#Offset_Int];
   #DummyBool := TRUE OR TRUE OR #StepSEQ_Pulse[#Offset_Int];
END_REGION

REGION Network 202: BLASTER #4 - Go to Skip_Exp4
   // Exceptions: 
   // 16#0000: Log(0) is not possible
   // 16#8000: Bit 15 is INT bit sign
   #_w1 := #NXT_SEQ_State = 16#0000;
   IF #_w1 THEN #FP_PARM.CurrentState[4] := 0; END_IF;
   #_w2 := #NXT_SEQ_State = 16#8000;
   IF #_w2 THEN #FP_PARM.CurrentState[4] := 16; END_IF;
   IF #_w1 OR #_w2 THEN GOTO Skip_Exp4; END_IF;
END_REGION

REGION Network 203: BLASTER #4 - Exponent of Step Mask Used as Step Number (for ECS Display)
   // Step Number = [ln(NXT_SEQ_State)/ln(2)]+1
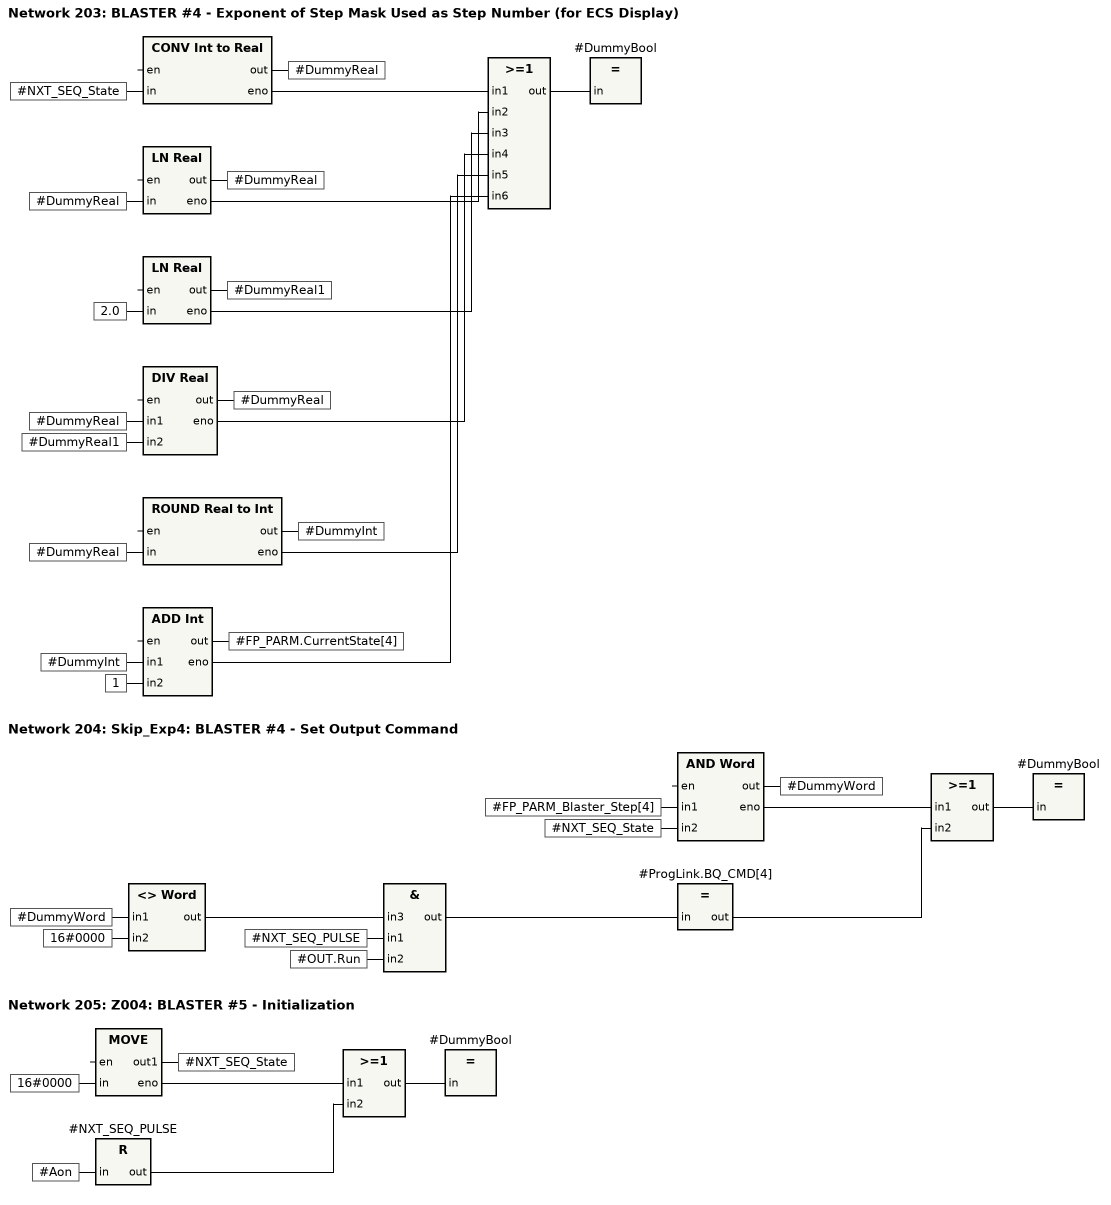
   #DummyReal := INT_TO_REAL(#NXT_SEQ_State);
   #DummyReal := LN(#DummyReal);
   #DummyReal1 := LN(2.0);
   #DummyReal := #DummyReal / #DummyReal1;
   #DummyInt := ROUND(#DummyReal);
   #FP_PARM.CurrentState[4] := #DummyInt + 1;
   #DummyBool := TRUE OR TRUE OR TRUE OR TRUE OR TRUE OR TRUE;
END_REGION

REGION Network 204: Skip_Exp4: BLASTER #4 - Set Output Command
   Skip_Exp4:
   #DummyWord := #FP_PARM_Blaster_Step[4] AND #NXT_SEQ_State;
   #ProgLink.BQ_CMD[4] := (#DummyWord <> 16#0000) AND #NXT_SEQ_PULSE AND #OUT.Run;
   #DummyBool := TRUE OR ((#DummyWord <> 16#0000) AND #NXT_SEQ_PULSE AND #OUT.Run);
END_REGION

REGION Network 205: Z004: BLASTER #5 - Initialization
   Z004:
   #NXT_SEQ_State := 16#0000;
   IF #Aon THEN #NXT_SEQ_PULSE := FALSE; END_IF;
   #DummyBool := TRUE OR #Aon;
END_REGION

REGION Network 206: BLASTER #5 - Go to Z005
   // If Blaster #5 is not configured in any sequence/step then clear state and go to next blaster
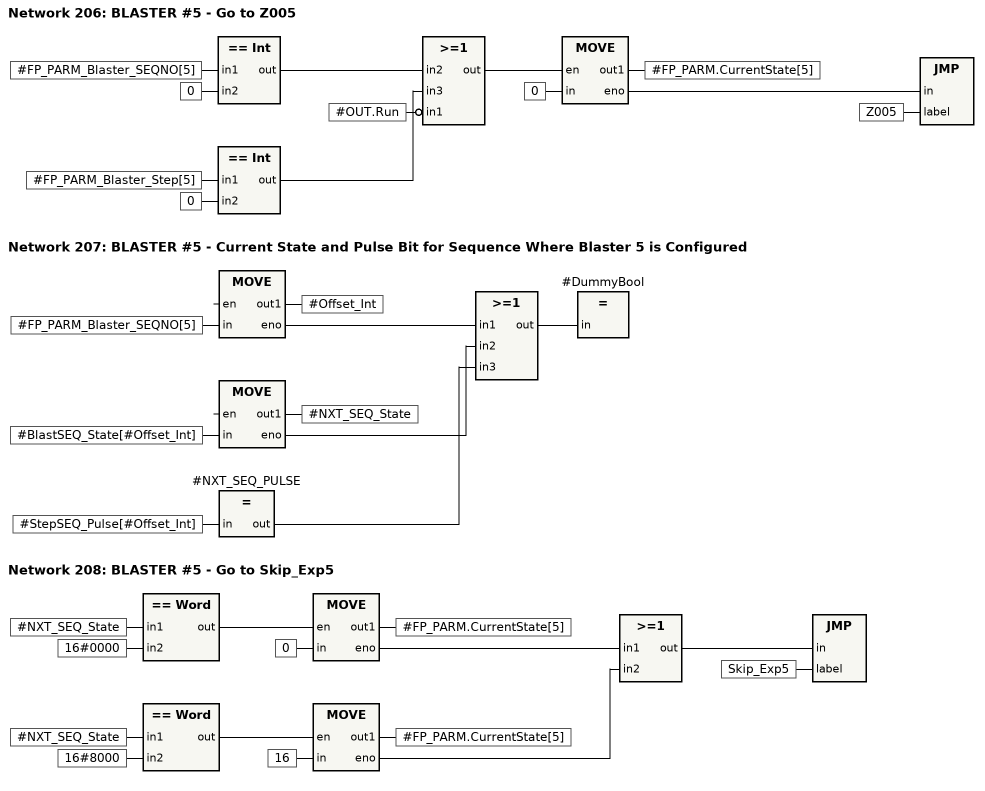
   #_w1 := (#FP_PARM_Blaster_SEQNO[5] = 0) OR (#FP_PARM_Blaster_Step[5] = 0) OR NOT #OUT.Run;
   IF #_w1 THEN
       #FP_PARM.CurrentState[5] := 0;
       GOTO Z005;
   END_IF;
END_REGION

REGION Network 207: BLASTER #5 - Current State and Pulse Bit for Sequence Where Blaster 5 is Configured
   #Offset_Int := #FP_PARM_Blaster_SEQNO[5];
   #NXT_SEQ_State := #BlastSEQ_State[#Offset_Int];
   #NXT_SEQ_PULSE := #StepSEQ_Pulse[#Offset_Int];
   #DummyBool := TRUE OR TRUE OR #StepSEQ_Pulse[#Offset_Int];
END_REGION

REGION Network 208: BLASTER #5 - Go to Skip_Exp5
   // Exceptions: 
   // 16#0000: Log(0) is not possible
   // 16#8000: Bit 15 is INT bit sign
   #_w1 := #NXT_SEQ_State = 16#0000;
   IF #_w1 THEN #FP_PARM.CurrentState[5] := 0; END_IF;
   #_w2 := #NXT_SEQ_State = 16#8000;
   IF #_w2 THEN #FP_PARM.CurrentState[5] := 16; END_IF;
   IF #_w1 OR #_w2 THEN GOTO Skip_Exp5; END_IF;
END_REGION

REGION Network 209: BLASTER #5 - Exponent of Step Mask Used as Step Number (for ECS Display)
   // Step Number = [ln(NXT_SEQ_State)/ln(2)]+1
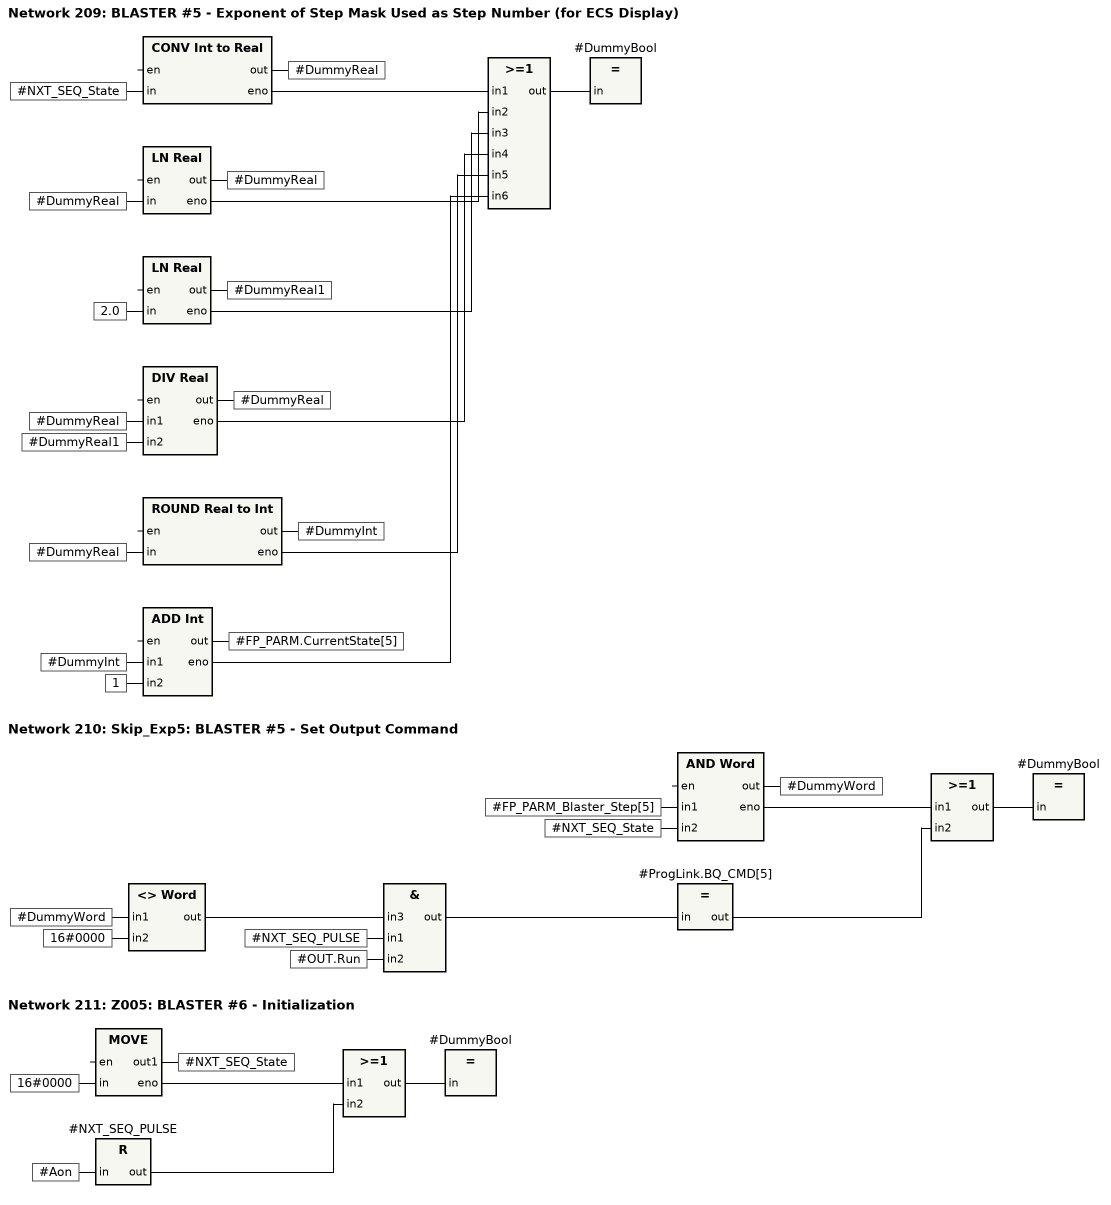
   #DummyReal := INT_TO_REAL(#NXT_SEQ_State);
   #DummyReal := LN(#DummyReal);
   #DummyReal1 := LN(2.0);
   #DummyReal := #DummyReal / #DummyReal1;
   #DummyInt := ROUND(#DummyReal);
   #FP_PARM.CurrentState[5] := #DummyInt + 1;
   #DummyBool := TRUE OR TRUE OR TRUE OR TRUE OR TRUE OR TRUE;
END_REGION

REGION Network 210: Skip_Exp5: BLASTER #5 - Set Output Command
   Skip_Exp5:
   #DummyWord := #FP_PARM_Blaster_Step[5] AND #NXT_SEQ_State;
   #ProgLink.BQ_CMD[5] := (#DummyWord <> 16#0000) AND #NXT_SEQ_PULSE AND #OUT.Run;
   #DummyBool := TRUE OR ((#DummyWord <> 16#0000) AND #NXT_SEQ_PULSE AND #OUT.Run);
END_REGION

REGION Network 211: Z005: BLASTER #6 - Initialization
   Z005:
   #NXT_SEQ_State := 16#0000;
   IF #Aon THEN #NXT_SEQ_PULSE := FALSE; END_IF;
   #DummyBool := TRUE OR #Aon;
END_REGION

REGION Network 212: BLASTER #6 - Go to Z006
   // If Blaster #6 is not configured in any sequence/step then clear state and go to next blaster
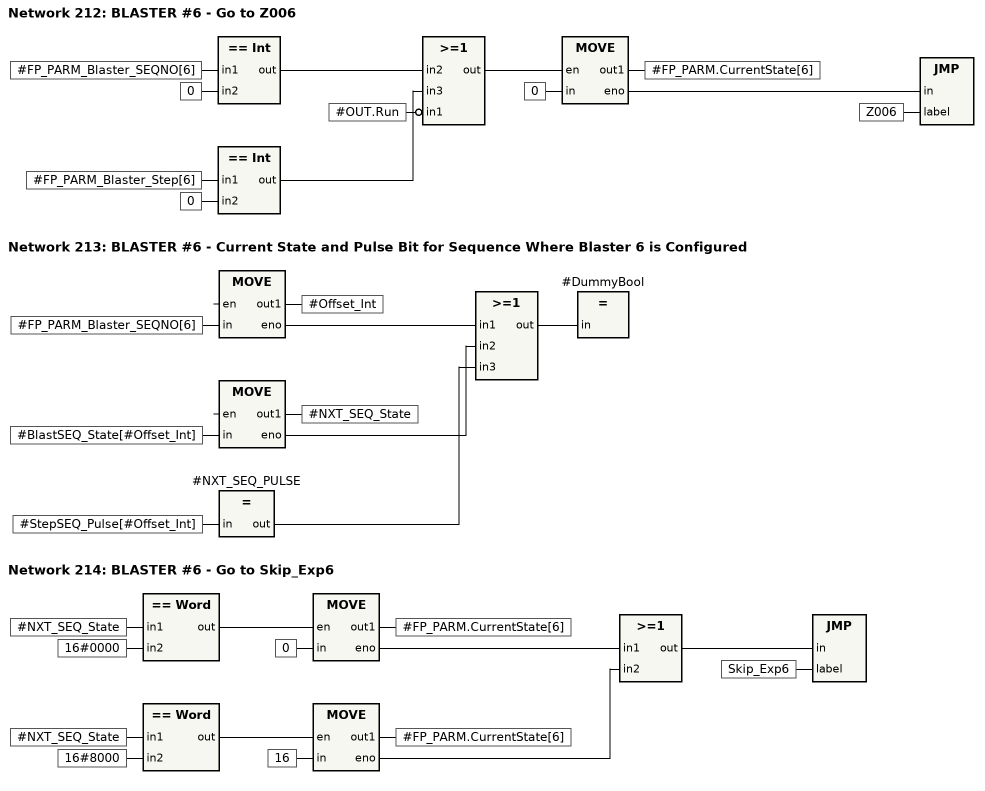
   #_w1 := (#FP_PARM_Blaster_SEQNO[6] = 0) OR (#FP_PARM_Blaster_Step[6] = 0) OR NOT #OUT.Run;
   IF #_w1 THEN
       #FP_PARM.CurrentState[6] := 0;
       GOTO Z006;
   END_IF;
END_REGION

REGION Network 213: BLASTER #6 - Current State and Pulse Bit for Sequence Where Blaster 6 is Configured
   #Offset_Int := #FP_PARM_Blaster_SEQNO[6];
   #NXT_SEQ_State := #BlastSEQ_State[#Offset_Int];
   #NXT_SEQ_PULSE := #StepSEQ_Pulse[#Offset_Int];
   #DummyBool := TRUE OR TRUE OR #StepSEQ_Pulse[#Offset_Int];
END_REGION

REGION Network 214: BLASTER #6 - Go to Skip_Exp6
   // Exceptions: 
   // 16#0000: Log(0) is not possible
   // 16#8000: Bit 15 is INT bit sign
   #_w1 := #NXT_SEQ_State = 16#0000;
   IF #_w1 THEN #FP_PARM.CurrentState[6] := 0; END_IF;
   #_w2 := #NXT_SEQ_State = 16#8000;
   IF #_w2 THEN #FP_PARM.CurrentState[6] := 16; END_IF;
   IF #_w1 OR #_w2 THEN GOTO Skip_Exp6; END_IF;
END_REGION

REGION Network 215: BLASTER #6 - Exponent of Step Mask Used as Step Number (for ECS Display)
   // Step Number = [ln(NXT_SEQ_State)/ln(2)]+1
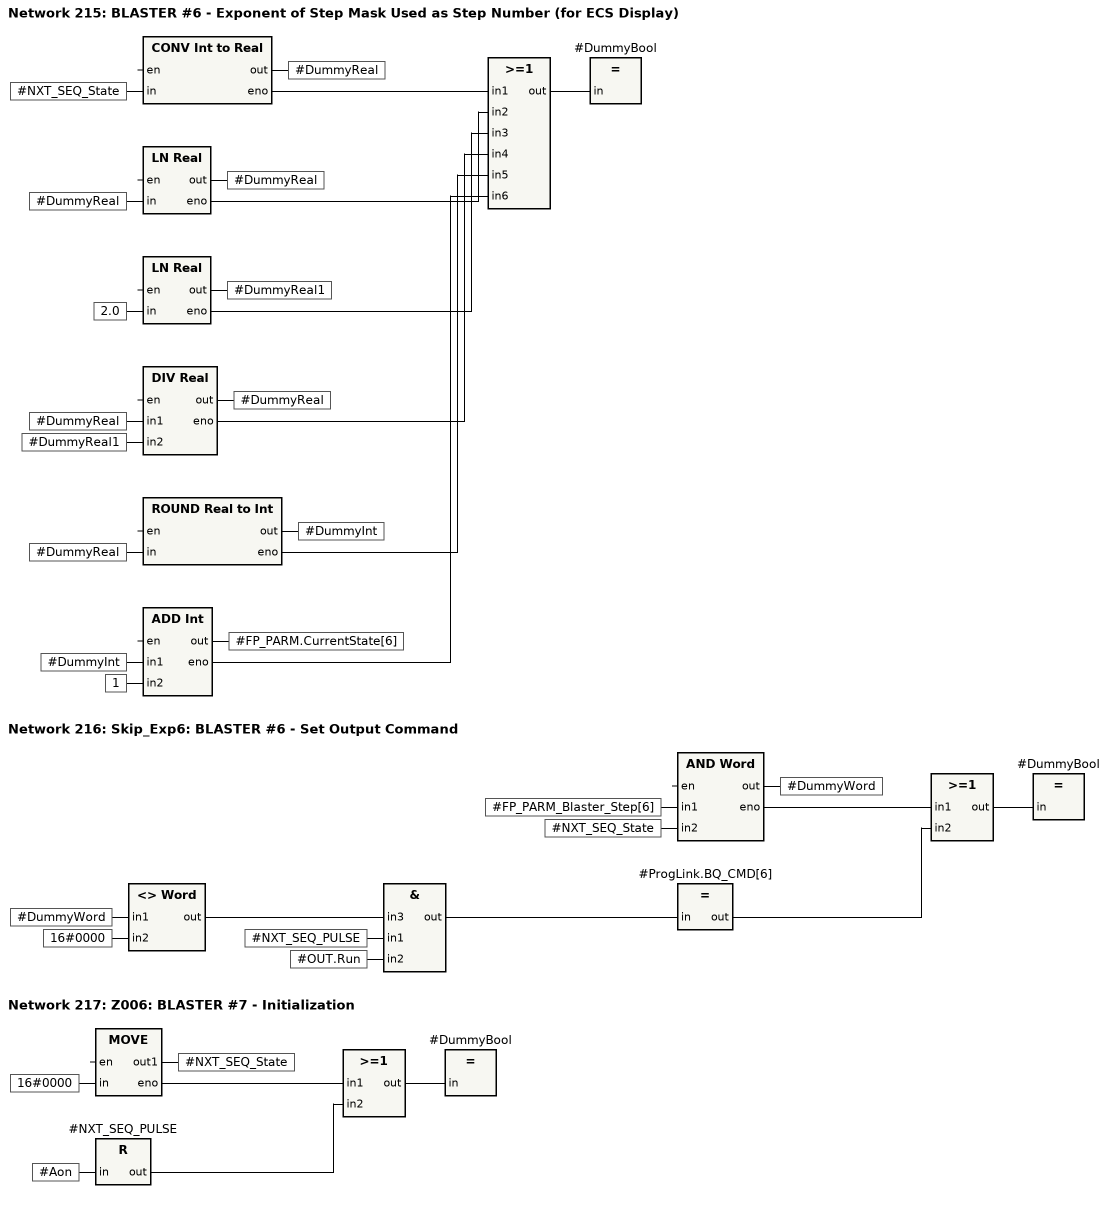
   #DummyReal := INT_TO_REAL(#NXT_SEQ_State);
   #DummyReal := LN(#DummyReal);
   #DummyReal1 := LN(2.0);
   #DummyReal := #DummyReal / #DummyReal1;
   #DummyInt := ROUND(#DummyReal);
   #FP_PARM.CurrentState[6] := #DummyInt + 1;
   #DummyBool := TRUE OR TRUE OR TRUE OR TRUE OR TRUE OR TRUE;
END_REGION

REGION Network 216: Skip_Exp6: BLASTER #6 - Set Output Command
   Skip_Exp6:
   #DummyWord := #FP_PARM_Blaster_Step[6] AND #NXT_SEQ_State;
   #ProgLink.BQ_CMD[6] := (#DummyWord <> 16#0000) AND #NXT_SEQ_PULSE AND #OUT.Run;
   #DummyBool := TRUE OR ((#DummyWord <> 16#0000) AND #NXT_SEQ_PULSE AND #OUT.Run);
END_REGION

REGION Network 217: Z006: BLASTER #7 - Initialization
   Z006:
   #NXT_SEQ_State := 16#0000;
   IF #Aon THEN #NXT_SEQ_PULSE := FALSE; END_IF;
   #DummyBool := TRUE OR #Aon;
END_REGION

REGION Network 218: BLASTER #7 - Go to Z007
   // If Blaster #7 is not configured in any sequence/step then clear state and go to next blaster
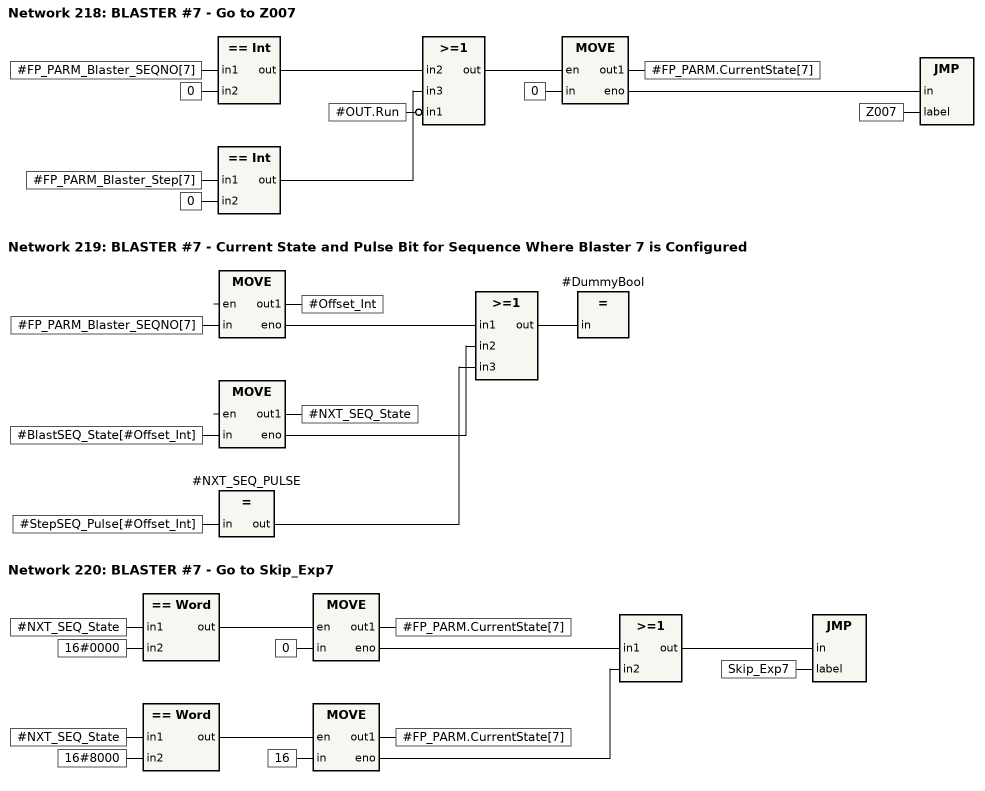
   #_w1 := (#FP_PARM_Blaster_SEQNO[7] = 0) OR (#FP_PARM_Blaster_Step[7] = 0) OR NOT #OUT.Run;
   IF #_w1 THEN
       #FP_PARM.CurrentState[7] := 0;
       GOTO Z007;
   END_IF;
END_REGION

REGION Network 219: BLASTER #7 - Current State and Pulse Bit for Sequence Where Blaster 7 is Configured
   #Offset_Int := #FP_PARM_Blaster_SEQNO[7];
   #NXT_SEQ_State := #BlastSEQ_State[#Offset_Int];
   #NXT_SEQ_PULSE := #StepSEQ_Pulse[#Offset_Int];
   #DummyBool := TRUE OR TRUE OR #StepSEQ_Pulse[#Offset_Int];
END_REGION

REGION Network 220: BLASTER #7 - Go to Skip_Exp7
   // Exceptions: 
   // 16#0000: Log(0) is not possible
   // 16#8000: Bit 15 is INT bit sign
   #_w1 := #NXT_SEQ_State = 16#0000;
   IF #_w1 THEN #FP_PARM.CurrentState[7] := 0; END_IF;
   #_w2 := #NXT_SEQ_State = 16#8000;
   IF #_w2 THEN #FP_PARM.CurrentState[7] := 16; END_IF;
   IF #_w1 OR #_w2 THEN GOTO Skip_Exp7; END_IF;
END_REGION

REGION Network 221: BLASTER #7 - Exponent of Step Mask Used as Step Number (for ECS Display)
   // Step Number = [ln(NXT_SEQ_State)/ln(2)]+1
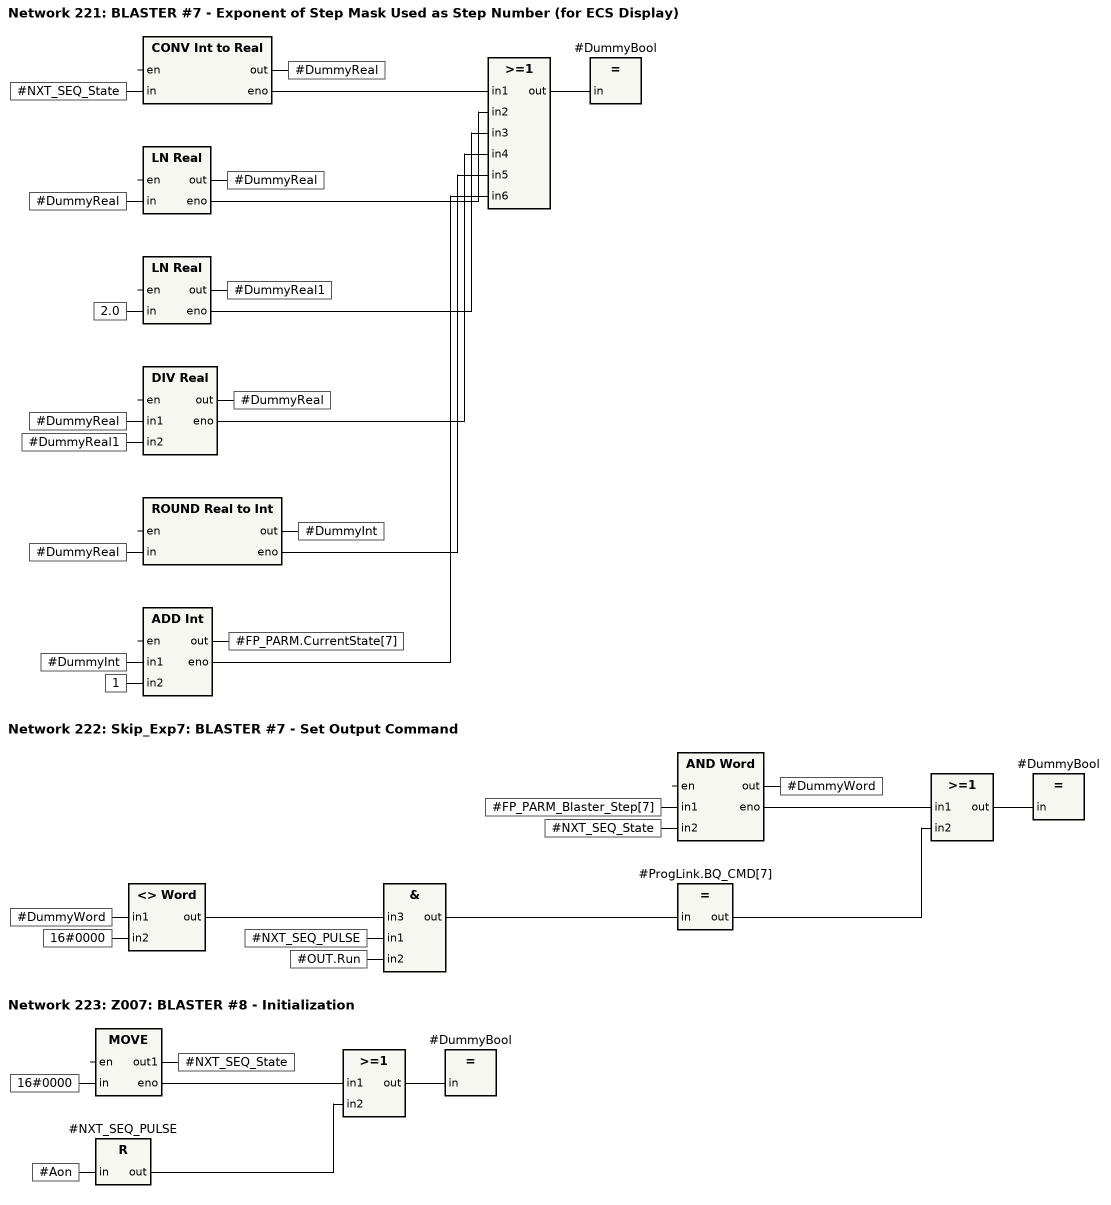
   #DummyReal := INT_TO_REAL(#NXT_SEQ_State);
   #DummyReal := LN(#DummyReal);
   #DummyReal1 := LN(2.0);
   #DummyReal := #DummyReal / #DummyReal1;
   #DummyInt := ROUND(#DummyReal);
   #FP_PARM.CurrentState[7] := #DummyInt + 1;
   #DummyBool := TRUE OR TRUE OR TRUE OR TRUE OR TRUE OR TRUE;
END_REGION

REGION Network 222: Skip_Exp7: BLASTER #7 - Set Output Command
   Skip_Exp7:
   #DummyWord := #FP_PARM_Blaster_Step[7] AND #NXT_SEQ_State;
   #ProgLink.BQ_CMD[7] := (#DummyWord <> 16#0000) AND #NXT_SEQ_PULSE AND #OUT.Run;
   #DummyBool := TRUE OR ((#DummyWord <> 16#0000) AND #NXT_SEQ_PULSE AND #OUT.Run);
END_REGION

REGION Network 223: Z007: BLASTER #8 - Initialization
   Z007:
   #NXT_SEQ_State := 16#0000;
   IF #Aon THEN #NXT_SEQ_PULSE := FALSE; END_IF;
   #DummyBool := TRUE OR #Aon;
END_REGION

REGION Network 224: BLASTER #8 - Go to Z008
   // If Blaster #8 is not configured in any sequence/step then clear state and go to next blaster
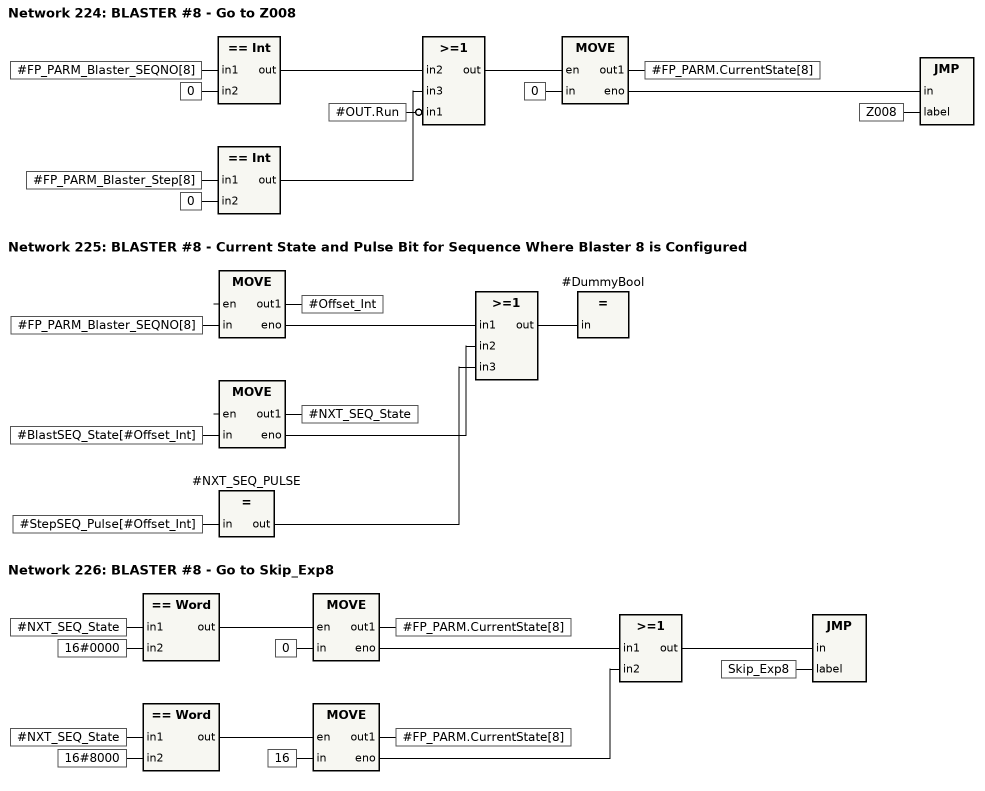
   #_w1 := (#FP_PARM_Blaster_SEQNO[8] = 0) OR (#FP_PARM_Blaster_Step[8] = 0) OR NOT #OUT.Run;
   IF #_w1 THEN
       #FP_PARM.CurrentState[8] := 0;
       GOTO Z008;
   END_IF;
END_REGION

REGION Network 225: BLASTER #8 - Current State and Pulse Bit for Sequence Where Blaster 8 is Configured
   #Offset_Int := #FP_PARM_Blaster_SEQNO[8];
   #NXT_SEQ_State := #BlastSEQ_State[#Offset_Int];
   #NXT_SEQ_PULSE := #StepSEQ_Pulse[#Offset_Int];
   #DummyBool := TRUE OR TRUE OR #StepSEQ_Pulse[#Offset_Int];
END_REGION

REGION Network 226: BLASTER #8 - Go to Skip_Exp8
   // Exceptions: 
   // 16#0000: Log(0) is not possible
   // 16#8000: Bit 15 is INT bit sign
   #_w1 := #NXT_SEQ_State = 16#0000;
   IF #_w1 THEN #FP_PARM.CurrentState[8] := 0; END_IF;
   #_w2 := #NXT_SEQ_State = 16#8000;
   IF #_w2 THEN #FP_PARM.CurrentState[8] := 16; END_IF;
   IF #_w1 OR #_w2 THEN GOTO Skip_Exp8; END_IF;
END_REGION

REGION Network 227: BLASTER #8 - Exponent of Step Mask Used as Step Number (for ECS Display)
   // Step Number = [ln(NXT_SEQ_State)/ln(2)]+1
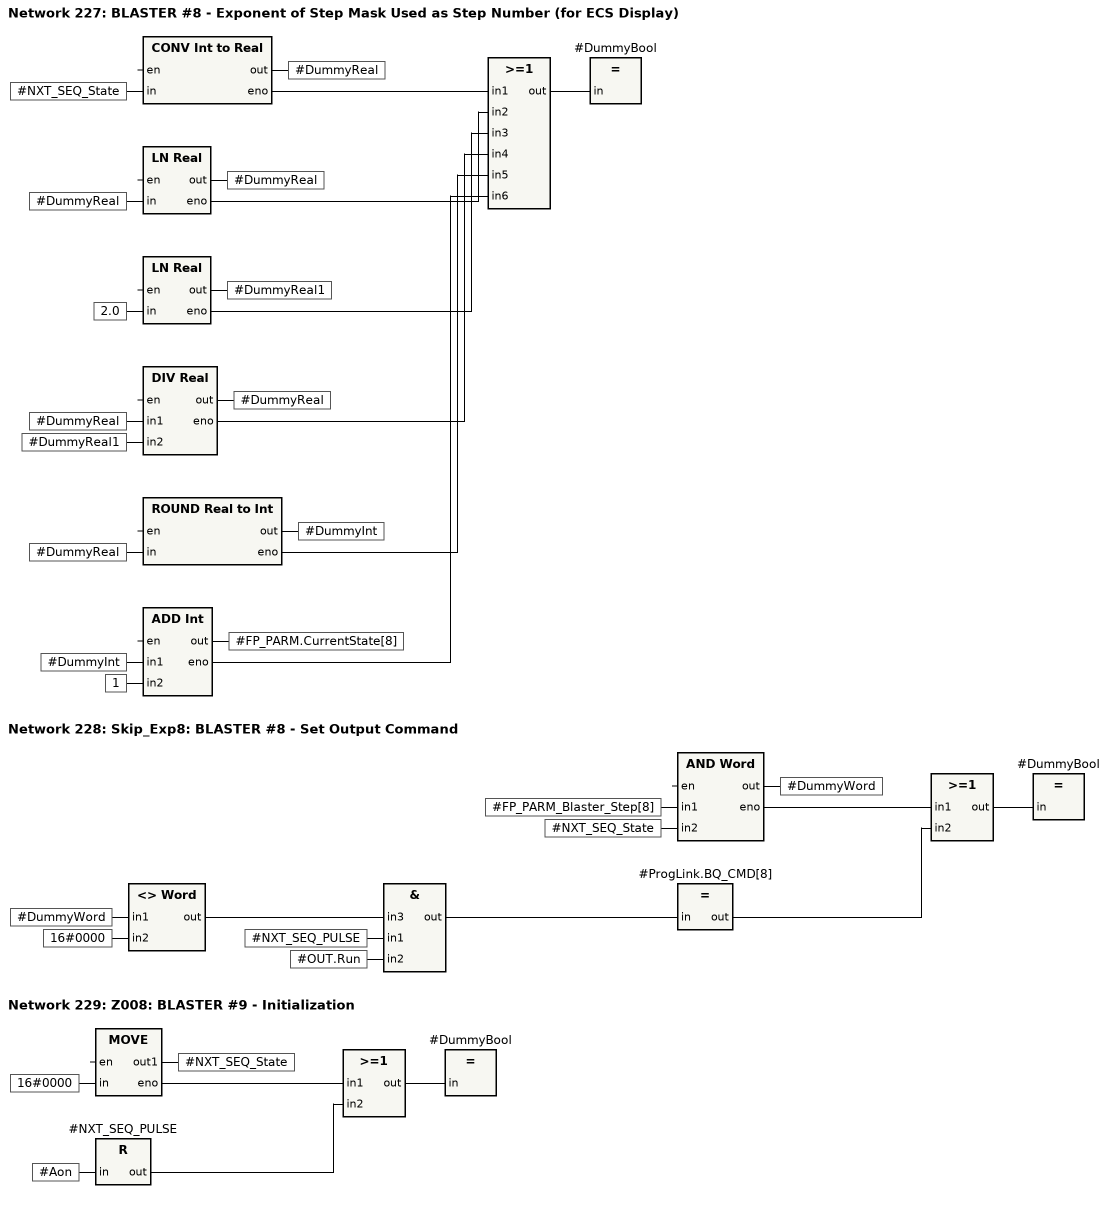
   #DummyReal := INT_TO_REAL(#NXT_SEQ_State);
   #DummyReal := LN(#DummyReal);
   #DummyReal1 := LN(2.0);
   #DummyReal := #DummyReal / #DummyReal1;
   #DummyInt := ROUND(#DummyReal);
   #FP_PARM.CurrentState[8] := #DummyInt + 1;
   #DummyBool := TRUE OR TRUE OR TRUE OR TRUE OR TRUE OR TRUE;
END_REGION

REGION Network 228: Skip_Exp8: BLASTER #8 - Set Output Command
   Skip_Exp8:
   #DummyWord := #FP_PARM_Blaster_Step[8] AND #NXT_SEQ_State;
   #ProgLink.BQ_CMD[8] := (#DummyWord <> 16#0000) AND #NXT_SEQ_PULSE AND #OUT.Run;
   #DummyBool := TRUE OR ((#DummyWord <> 16#0000) AND #NXT_SEQ_PULSE AND #OUT.Run);
END_REGION

REGION Network 229: Z008: BLASTER #9 - Initialization
   Z008:
   #NXT_SEQ_State := 16#0000;
   IF #Aon THEN #NXT_SEQ_PULSE := FALSE; END_IF;
   #DummyBool := TRUE OR #Aon;
END_REGION

REGION Network 230: BLASTER #9 - Go to Z009
   // If Blaster #9 is not configured in any sequence/step then clear state and go to next blaster
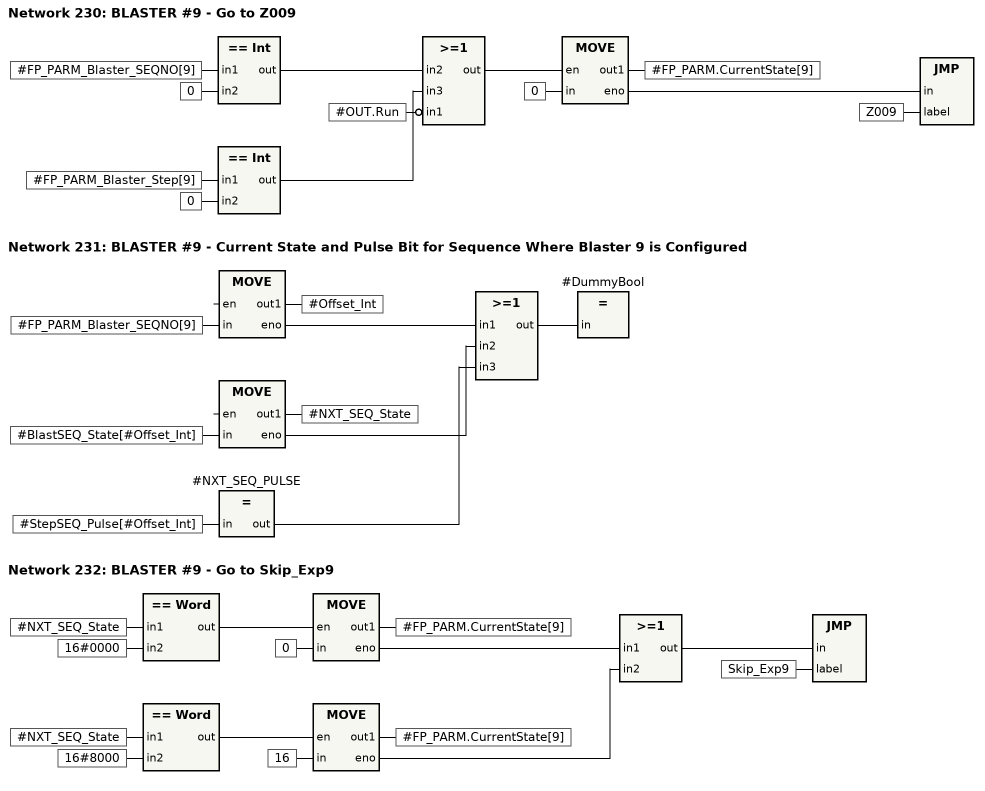
   #_w1 := (#FP_PARM_Blaster_SEQNO[9] = 0) OR (#FP_PARM_Blaster_Step[9] = 0) OR NOT #OUT.Run;
   IF #_w1 THEN
       #FP_PARM.CurrentState[9] := 0;
       GOTO Z009;
   END_IF;
END_REGION

REGION Network 231: BLASTER #9 - Current State and Pulse Bit for Sequence Where Blaster 9 is Configured
   #Offset_Int := #FP_PARM_Blaster_SEQNO[9];
   #NXT_SEQ_State := #BlastSEQ_State[#Offset_Int];
   #NXT_SEQ_PULSE := #StepSEQ_Pulse[#Offset_Int];
   #DummyBool := TRUE OR TRUE OR #StepSEQ_Pulse[#Offset_Int];
END_REGION

REGION Network 232: BLASTER #9 - Go to Skip_Exp9
   // Exceptions: 
   // 16#0000: Log(0) is not possible
   // 16#8000: Bit 15 is INT bit sign
   #_w1 := #NXT_SEQ_State = 16#0000;
   IF #_w1 THEN #FP_PARM.CurrentState[9] := 0; END_IF;
   #_w2 := #NXT_SEQ_State = 16#8000;
   IF #_w2 THEN #FP_PARM.CurrentState[9] := 16; END_IF;
   IF #_w1 OR #_w2 THEN GOTO Skip_Exp9; END_IF;
END_REGION

REGION Network 233: BLASTER #9 - Exponent of Step Mask Used as Step Number (for ECS Display)
   // Step Number = [ln(NXT_SEQ_State)/ln(2)]+1
